REGION Network 64: Step[1390] : Job[13] Step End
   RUNG wire#powerrail
      { S7_Templates := "SrcType := DInt" } EQ_Contact(in1 := "Unit1.Em5.ControlNodes".gaugeRnR.sequence.status.currentStep, in2 := #JOB_13_STEP_90)
      Contact( "Unit1.Em5.ControlNodes".gaugeRnR.sequence.status.seqActive )
      wire#w1
      Coil( "Unit1.Em5.ControlNodes".gaugeRnR."step".action1[1390] )
   END_RUNG
   RUNG wire#w1
      Coil( "Unit1.Em5.ControlNodes".gaugeRnR."step".transition1[1390] )
   END_RUNG
   RUNG wire#w1
      Contact( "Unit1.Em5.ControlNodes".gaugeRnR."step".transition1[1390] )
      Move(in := #STEP_IDLE, out1 => "Unit1.Em5.ControlNodes".gaugeRnR.sequence.status.nextStep)
   END_RUNG
   // the same network as SCL:
   "Unit1.Em5.ControlNodes".gaugeRnR."step".action1[1390] := ("Unit1.Em5.ControlNodes".gaugeRnR.sequence.status.currentStep = #JOB_13_STEP_90) AND "Unit1.Em5.ControlNodes".gaugeRnR.sequence.status.seqActive;
   "Unit1.Em5.ControlNodes".gaugeRnR."step".transition1[1390] := ("Unit1.Em5.ControlNodes".gaugeRnR.sequence.status.currentStep = #JOB_13_STEP_90) AND "Unit1.Em5.ControlNodes".gaugeRnR.sequence.status.seqActive;
   IF ("Unit1.Em5.ControlNodes".gaugeRnR.sequence.status.currentStep = #JOB_13_STEP_90) AND "Unit1.Em5.ControlNodes".gaugeRnR.sequence.status.seqActive AND "Unit1.Em5.ControlNodes".gaugeRnR."step".transition1[1390] THEN
       "Unit1.Em5.ControlNodes".gaugeRnR.sequence.status.nextStep := #STEP_IDLE;
   END_IF;
END_REGION

REGION Network 65: *************** JOB[15] MainPnP Move ReelCut Convyeor / AlignTable************************
END_REGION

REGION Network 66: Step[1501] : Job[15] Condtion
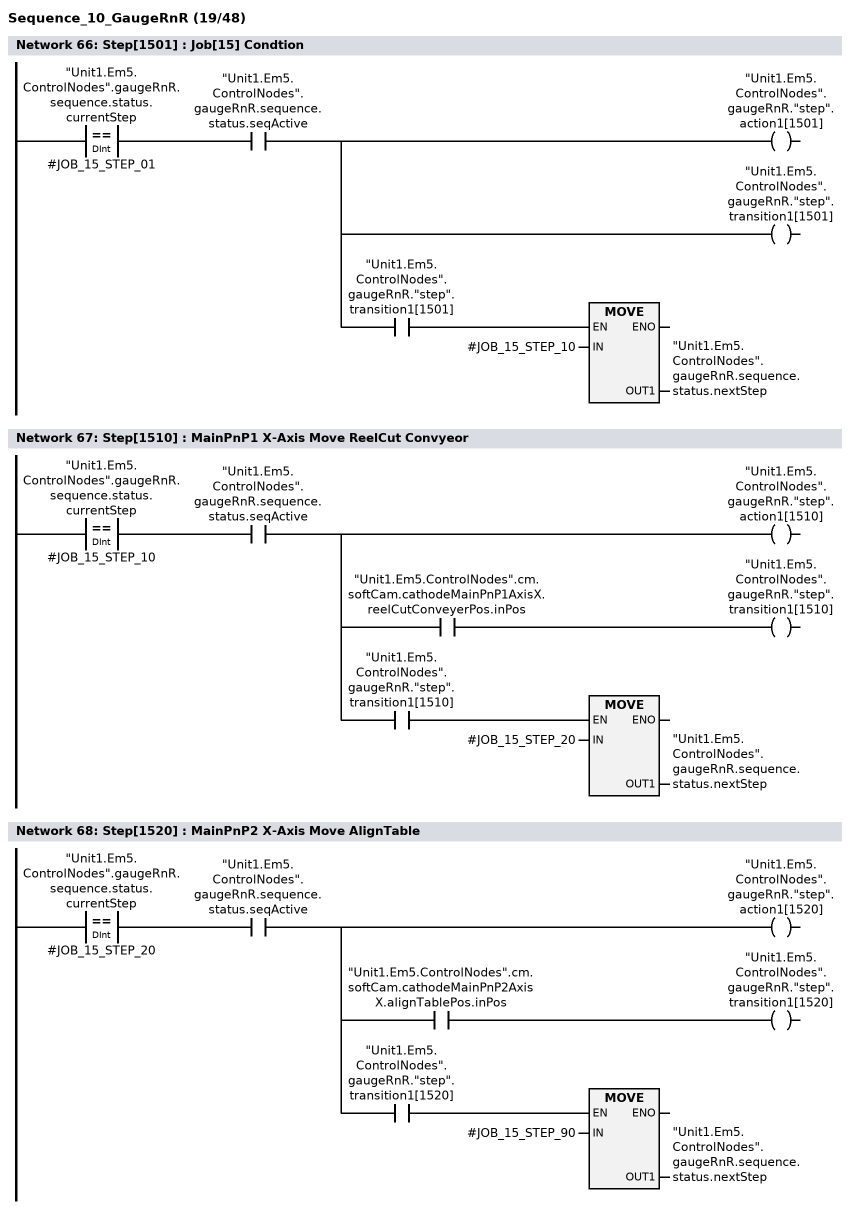
   RUNG wire#powerrail
      { S7_Templates := "SrcType := DInt" } EQ_Contact(in1 := "Unit1.Em5.ControlNodes".gaugeRnR.sequence.status.currentStep, in2 := #JOB_15_STEP_01)
      Contact( "Unit1.Em5.ControlNodes".gaugeRnR.sequence.status.seqActive )
      wire#w1
      Coil( "Unit1.Em5.ControlNodes".gaugeRnR."step".action1[1501] )
   END_RUNG
   RUNG wire#w1
      Coil( "Unit1.Em5.ControlNodes".gaugeRnR."step".transition1[1501] )
   END_RUNG
   RUNG wire#w1
      Contact( "Unit1.Em5.ControlNodes".gaugeRnR."step".transition1[1501] )
      Move(in := #JOB_15_STEP_10, out1 => "Unit1.Em5.ControlNodes".gaugeRnR.sequence.status.nextStep)
   END_RUNG
   // the same network as SCL:
   "Unit1.Em5.ControlNodes".gaugeRnR."step".action1[1501] := ("Unit1.Em5.ControlNodes".gaugeRnR.sequence.status.currentStep = #JOB_15_STEP_01) AND "Unit1.Em5.ControlNodes".gaugeRnR.sequence.status.seqActive;
   "Unit1.Em5.ControlNodes".gaugeRnR."step".transition1[1501] := ("Unit1.Em5.ControlNodes".gaugeRnR.sequence.status.currentStep = #JOB_15_STEP_01) AND "Unit1.Em5.ControlNodes".gaugeRnR.sequence.status.seqActive;
   IF ("Unit1.Em5.ControlNodes".gaugeRnR.sequence.status.currentStep = #JOB_15_STEP_01) AND "Unit1.Em5.ControlNodes".gaugeRnR.sequence.status.seqActive AND "Unit1.Em5.ControlNodes".gaugeRnR."step".transition1[1501] THEN
       "Unit1.Em5.ControlNodes".gaugeRnR.sequence.status.nextStep := #JOB_15_STEP_10;
   END_IF;
END_REGION

REGION Network 67: Step[1510] : MainPnP1 X-Axis Move ReelCut Convyeor
   RUNG wire#powerrail
      { S7_Templates := "SrcType := DInt" } EQ_Contact(in1 := "Unit1.Em5.ControlNodes".gaugeRnR.sequence.status.currentStep, in2 := #JOB_15_STEP_10)
      Contact( "Unit1.Em5.ControlNodes".gaugeRnR.sequence.status.seqActive )
      wire#w1
      Coil( "Unit1.Em5.ControlNodes".gaugeRnR."step".action1[1510] )
   END_RUNG
   RUNG wire#w1
      Contact( "Unit1.Em5.ControlNodes".cm.softCam.cathodeMainPnP1AxisX.reelCutConveyerPos.inPos )
      Coil( "Unit1.Em5.ControlNodes".gaugeRnR."step".transition1[1510] )
   END_RUNG
   RUNG wire#w1
      Contact( "Unit1.Em5.ControlNodes".gaugeRnR."step".transition1[1510] )
      Move(in := #JOB_15_STEP_20, out1 => "Unit1.Em5.ControlNodes".gaugeRnR.sequence.status.nextStep)
   END_RUNG
   // the same network as SCL:
   "Unit1.Em5.ControlNodes".gaugeRnR."step".action1[1510] := ("Unit1.Em5.ControlNodes".gaugeRnR.sequence.status.currentStep = #JOB_15_STEP_10) AND "Unit1.Em5.ControlNodes".gaugeRnR.sequence.status.seqActive;
   "Unit1.Em5.ControlNodes".gaugeRnR."step".transition1[1510] := ("Unit1.Em5.ControlNodes".gaugeRnR.sequence.status.currentStep = #JOB_15_STEP_10) AND "Unit1.Em5.ControlNodes".gaugeRnR.sequence.status.seqActive AND "Unit1.Em5.ControlNodes".cm.softCam.cathodeMainPnP1AxisX.reelCutConveyerPos.inPos;
   IF ("Unit1.Em5.ControlNodes".gaugeRnR.sequence.status.currentStep = #JOB_15_STEP_10) AND "Unit1.Em5.ControlNodes".gaugeRnR.sequence.status.seqActive AND "Unit1.Em5.ControlNodes".gaugeRnR."step".transition1[1510] THEN
       "Unit1.Em5.ControlNodes".gaugeRnR.sequence.status.nextStep := #JOB_15_STEP_20;
   END_IF;
END_REGION

REGION Network 68: Step[1520] : MainPnP2 X-Axis Move AlignTable
   RUNG wire#powerrail
      { S7_Templates := "SrcType := DInt" } EQ_Contact(in1 := "Unit1.Em5.ControlNodes".gaugeRnR.sequence.status.currentStep, in2 := #JOB_15_STEP_20)
      Contact( "Unit1.Em5.ControlNodes".gaugeRnR.sequence.status.seqActive )
      wire#w1
      Coil( "Unit1.Em5.ControlNodes".gaugeRnR."step".action1[1520] )
   END_RUNG
   RUNG wire#w1
      Contact( "Unit1.Em5.ControlNodes".cm.softCam.cathodeMainPnP2AxisX.alignTablePos.inPos )
      Coil( "Unit1.Em5.ControlNodes".gaugeRnR."step".transition1[1520] )
   END_RUNG
   RUNG wire#w1
      Contact( "Unit1.Em5.ControlNodes".gaugeRnR."step".transition1[1520] )
      Move(in := #JOB_15_STEP_90, out1 => "Unit1.Em5.ControlNodes".gaugeRnR.sequence.status.nextStep)
   END_RUNG
   // the same network as SCL:
   "Unit1.Em5.ControlNodes".gaugeRnR."step".action1[1520] := ("Unit1.Em5.ControlNodes".gaugeRnR.sequence.status.currentStep = #JOB_15_STEP_20) AND "Unit1.Em5.ControlNodes".gaugeRnR.sequence.status.seqActive;
   "Unit1.Em5.ControlNodes".gaugeRnR."step".transition1[1520] := ("Unit1.Em5.ControlNodes".gaugeRnR.sequence.status.currentStep = #JOB_15_STEP_20) AND "Unit1.Em5.ControlNodes".gaugeRnR.sequence.status.seqActive AND "Unit1.Em5.ControlNodes".cm.softCam.cathodeMainPnP2AxisX.alignTablePos.inPos;
   IF ("Unit1.Em5.ControlNodes".gaugeRnR.sequence.status.currentStep = #JOB_15_STEP_20) AND "Unit1.Em5.ControlNodes".gaugeRnR.sequence.status.seqActive AND "Unit1.Em5.ControlNodes".gaugeRnR."step".transition1[1520] THEN
       "Unit1.Em5.ControlNodes".gaugeRnR.sequence.status.nextStep := #JOB_15_STEP_90;
   END_IF;
END_REGION

REGION Network 69: Step[1590] : Job[15] Step End
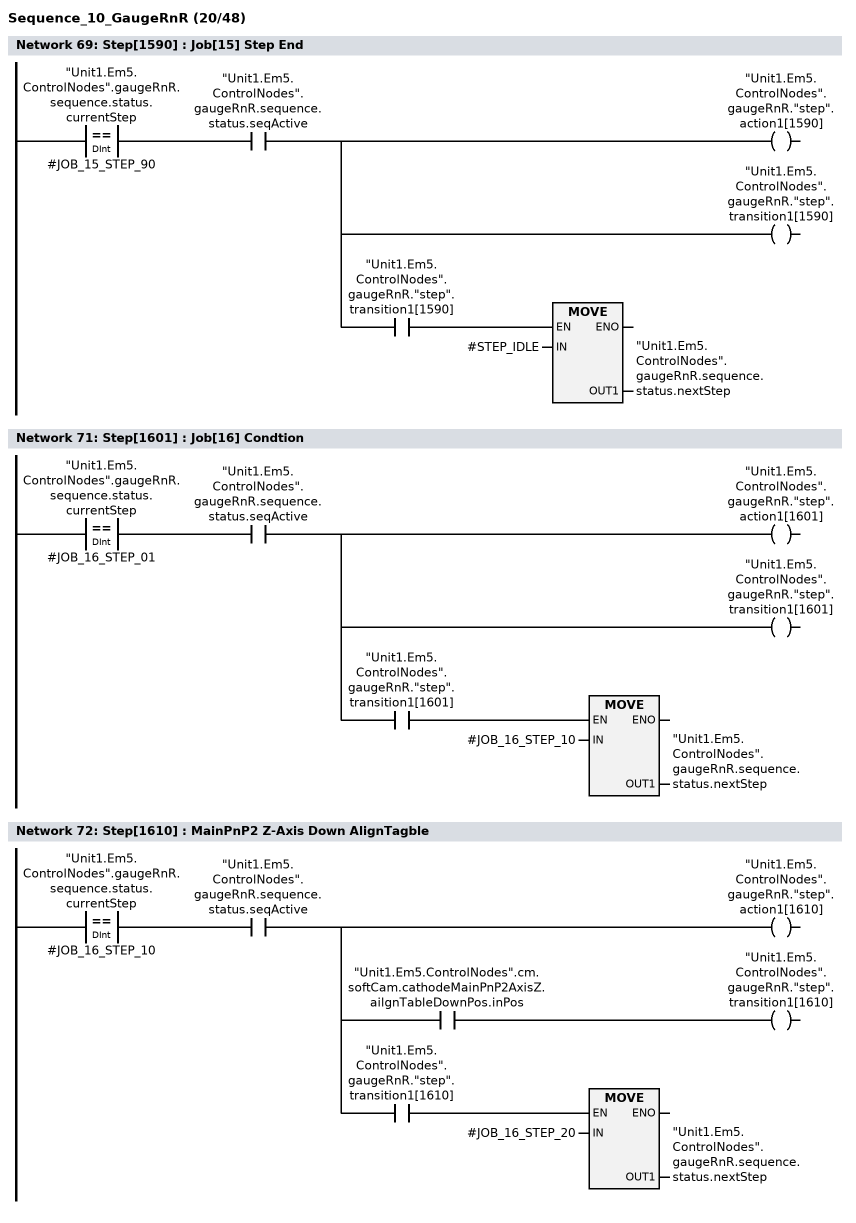
   RUNG wire#powerrail
      { S7_Templates := "SrcType := DInt" } EQ_Contact(in1 := "Unit1.Em5.ControlNodes".gaugeRnR.sequence.status.currentStep, in2 := #JOB_15_STEP_90)
      Contact( "Unit1.Em5.ControlNodes".gaugeRnR.sequence.status.seqActive )
      wire#w1
      Coil( "Unit1.Em5.ControlNodes".gaugeRnR."step".action1[1590] )
   END_RUNG
   RUNG wire#w1
      Coil( "Unit1.Em5.ControlNodes".gaugeRnR."step".transition1[1590] )
   END_RUNG
   RUNG wire#w1
      Contact( "Unit1.Em5.ControlNodes".gaugeRnR."step".transition1[1590] )
      Move(in := #STEP_IDLE, out1 => "Unit1.Em5.ControlNodes".gaugeRnR.sequence.status.nextStep)
   END_RUNG
   // the same network as SCL:
   "Unit1.Em5.ControlNodes".gaugeRnR."step".action1[1590] := ("Unit1.Em5.ControlNodes".gaugeRnR.sequence.status.currentStep = #JOB_15_STEP_90) AND "Unit1.Em5.ControlNodes".gaugeRnR.sequence.status.seqActive;
   "Unit1.Em5.ControlNodes".gaugeRnR."step".transition1[1590] := ("Unit1.Em5.ControlNodes".gaugeRnR.sequence.status.currentStep = #JOB_15_STEP_90) AND "Unit1.Em5.ControlNodes".gaugeRnR.sequence.status.seqActive;
   IF ("Unit1.Em5.ControlNodes".gaugeRnR.sequence.status.currentStep = #JOB_15_STEP_90) AND "Unit1.Em5.ControlNodes".gaugeRnR.sequence.status.seqActive AND "Unit1.Em5.ControlNodes".gaugeRnR."step".transition1[1590] THEN
       "Unit1.Em5.ControlNodes".gaugeRnR.sequence.status.nextStep := #STEP_IDLE;
   END_IF;
END_REGION

REGION Network 70: *************** JOB[16] AlignTable To MainPnP2 ************************
END_REGION

REGION Network 71: Step[1601] : Job[16] Condtion
   RUNG wire#powerrail
      { S7_Templates := "SrcType := DInt" } EQ_Contact(in1 := "Unit1.Em5.ControlNodes".gaugeRnR.sequence.status.currentStep, in2 := #JOB_16_STEP_01)
      Contact( "Unit1.Em5.ControlNodes".gaugeRnR.sequence.status.seqActive )
      wire#w1
      Coil( "Unit1.Em5.ControlNodes".gaugeRnR."step".action1[1601] )
   END_RUNG
   RUNG wire#w1
      Coil( "Unit1.Em5.ControlNodes".gaugeRnR."step".transition1[1601] )
   END_RUNG
   RUNG wire#w1
      Contact( "Unit1.Em5.ControlNodes".gaugeRnR."step".transition1[1601] )
      Move(in := #JOB_16_STEP_10, out1 => "Unit1.Em5.ControlNodes".gaugeRnR.sequence.status.nextStep)
   END_RUNG
   // the same network as SCL:
   "Unit1.Em5.ControlNodes".gaugeRnR."step".action1[1601] := ("Unit1.Em5.ControlNodes".gaugeRnR.sequence.status.currentStep = #JOB_16_STEP_01) AND "Unit1.Em5.ControlNodes".gaugeRnR.sequence.status.seqActive;
   "Unit1.Em5.ControlNodes".gaugeRnR."step".transition1[1601] := ("Unit1.Em5.ControlNodes".gaugeRnR.sequence.status.currentStep = #JOB_16_STEP_01) AND "Unit1.Em5.ControlNodes".gaugeRnR.sequence.status.seqActive;
   IF ("Unit1.Em5.ControlNodes".gaugeRnR.sequence.status.currentStep = #JOB_16_STEP_01) AND "Unit1.Em5.ControlNodes".gaugeRnR.sequence.status.seqActive AND "Unit1.Em5.ControlNodes".gaugeRnR."step".transition1[1601] THEN
       "Unit1.Em5.ControlNodes".gaugeRnR.sequence.status.nextStep := #JOB_16_STEP_10;
   END_IF;
END_REGION

REGION Network 72: Step[1610] : MainPnP2 Z-Axis Down AlignTagble
   RUNG wire#powerrail
      { S7_Templates := "SrcType := DInt" } EQ_Contact(in1 := "Unit1.Em5.ControlNodes".gaugeRnR.sequence.status.currentStep, in2 := #JOB_16_STEP_10)
      Contact( "Unit1.Em5.ControlNodes".gaugeRnR.sequence.status.seqActive )
      wire#w1
      Coil( "Unit1.Em5.ControlNodes".gaugeRnR."step".action1[1610] )
   END_RUNG
   RUNG wire#w1
      Contact( "Unit1.Em5.ControlNodes".cm.softCam.cathodeMainPnP2AxisZ.ailgnTableDownPos.inPos )
      Coil( "Unit1.Em5.ControlNodes".gaugeRnR."step".transition1[1610] )
   END_RUNG
   RUNG wire#w1
      Contact( "Unit1.Em5.ControlNodes".gaugeRnR."step".transition1[1610] )
      Move(in := #JOB_16_STEP_20, out1 => "Unit1.Em5.ControlNodes".gaugeRnR.sequence.status.nextStep)
   END_RUNG
   // the same network as SCL:
   "Unit1.Em5.ControlNodes".gaugeRnR."step".action1[1610] := ("Unit1.Em5.ControlNodes".gaugeRnR.sequence.status.currentStep = #JOB_16_STEP_10) AND "Unit1.Em5.ControlNodes".gaugeRnR.sequence.status.seqActive;
   "Unit1.Em5.ControlNodes".gaugeRnR."step".transition1[1610] := ("Unit1.Em5.ControlNodes".gaugeRnR.sequence.status.currentStep = #JOB_16_STEP_10) AND "Unit1.Em5.ControlNodes".gaugeRnR.sequence.status.seqActive AND "Unit1.Em5.ControlNodes".cm.softCam.cathodeMainPnP2AxisZ.ailgnTableDownPos.inPos;
   IF ("Unit1.Em5.ControlNodes".gaugeRnR.sequence.status.currentStep = #JOB_16_STEP_10) AND "Unit1.Em5.ControlNodes".gaugeRnR.sequence.status.seqActive AND "Unit1.Em5.ControlNodes".gaugeRnR."step".transition1[1610] THEN
       "Unit1.Em5.ControlNodes".gaugeRnR.sequence.status.nextStep := #JOB_16_STEP_20;
   END_IF;
END_REGION

REGION Network 73: Step[1620] : AlignTable Vaccum Off
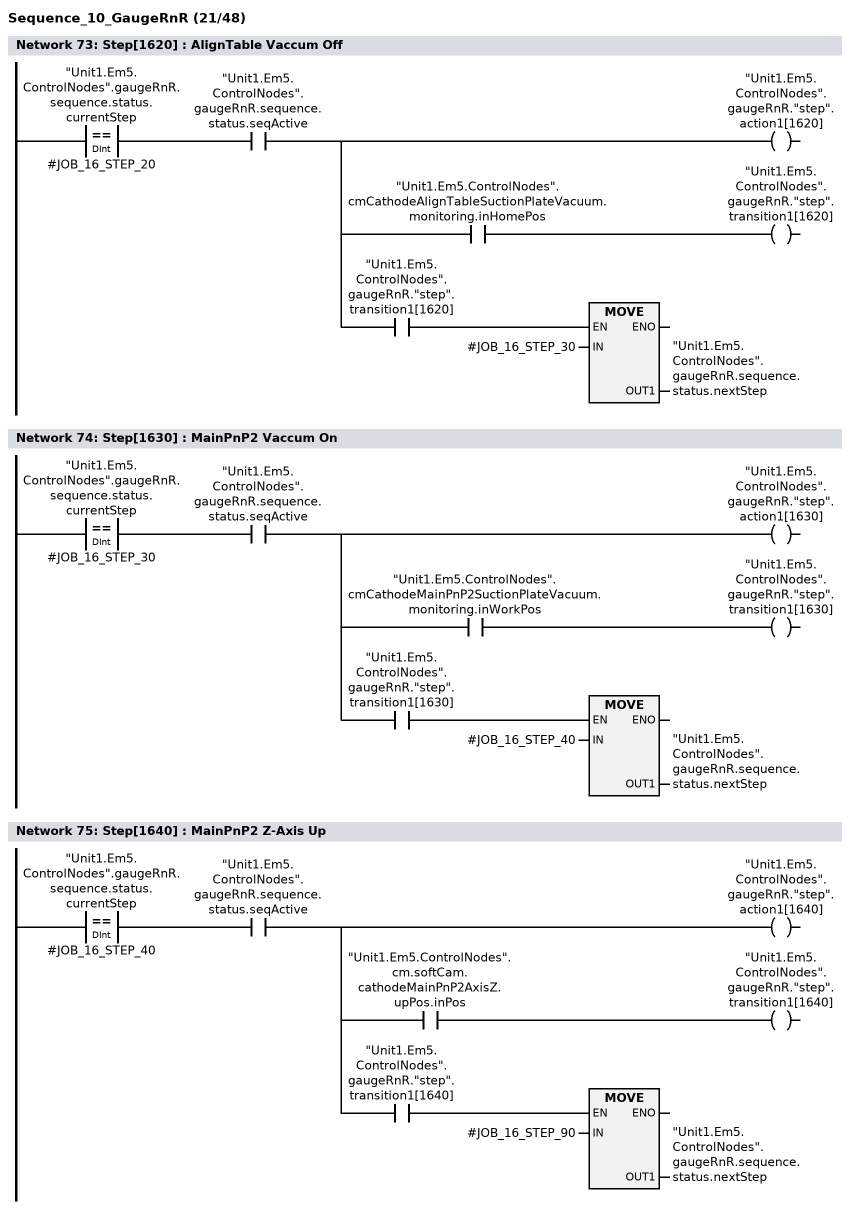
   RUNG wire#powerrail
      { S7_Templates := "SrcType := DInt" } EQ_Contact(in1 := "Unit1.Em5.ControlNodes".gaugeRnR.sequence.status.currentStep, in2 := #JOB_16_STEP_20)
      Contact( "Unit1.Em5.ControlNodes".gaugeRnR.sequence.status.seqActive )
      wire#w1
      Coil( "Unit1.Em5.ControlNodes".gaugeRnR."step".action1[1620] )
   END_RUNG
   RUNG wire#w1
      Contact( "Unit1.Em5.ControlNodes".cmCathodeAlignTableSuctionPlateVacuum.monitoring.inHomePos )
      Coil( "Unit1.Em5.ControlNodes".gaugeRnR."step".transition1[1620] )
   END_RUNG
   RUNG wire#w1
      Contact( "Unit1.Em5.ControlNodes".gaugeRnR."step".transition1[1620] )
      Move(in := #JOB_16_STEP_30, out1 => "Unit1.Em5.ControlNodes".gaugeRnR.sequence.status.nextStep)
   END_RUNG
   // the same network as SCL:
   "Unit1.Em5.ControlNodes".gaugeRnR."step".action1[1620] := ("Unit1.Em5.ControlNodes".gaugeRnR.sequence.status.currentStep = #JOB_16_STEP_20) AND "Unit1.Em5.ControlNodes".gaugeRnR.sequence.status.seqActive;
   "Unit1.Em5.ControlNodes".gaugeRnR."step".transition1[1620] := ("Unit1.Em5.ControlNodes".gaugeRnR.sequence.status.currentStep = #JOB_16_STEP_20) AND "Unit1.Em5.ControlNodes".gaugeRnR.sequence.status.seqActive AND "Unit1.Em5.ControlNodes".cmCathodeAlignTableSuctionPlateVacuum.monitoring.inHomePos;
   IF ("Unit1.Em5.ControlNodes".gaugeRnR.sequence.status.currentStep = #JOB_16_STEP_20) AND "Unit1.Em5.ControlNodes".gaugeRnR.sequence.status.seqActive AND "Unit1.Em5.ControlNodes".gaugeRnR."step".transition1[1620] THEN
       "Unit1.Em5.ControlNodes".gaugeRnR.sequence.status.nextStep := #JOB_16_STEP_30;
   END_IF;
END_REGION

REGION Network 74: Step[1630] : MainPnP2 Vaccum On
   RUNG wire#powerrail
      { S7_Templates := "SrcType := DInt" } EQ_Contact(in1 := "Unit1.Em5.ControlNodes".gaugeRnR.sequence.status.currentStep, in2 := #JOB_16_STEP_30)
      Contact( "Unit1.Em5.ControlNodes".gaugeRnR.sequence.status.seqActive )
      wire#w1
      Coil( "Unit1.Em5.ControlNodes".gaugeRnR."step".action1[1630] )
   END_RUNG
   RUNG wire#w1
      Contact( "Unit1.Em5.ControlNodes".cmCathodeMainPnP2SuctionPlateVacuum.monitoring.inWorkPos )
      Coil( "Unit1.Em5.ControlNodes".gaugeRnR."step".transition1[1630] )
   END_RUNG
   RUNG wire#w1
      Contact( "Unit1.Em5.ControlNodes".gaugeRnR."step".transition1[1630] )
      Move(in := #JOB_16_STEP_40, out1 => "Unit1.Em5.ControlNodes".gaugeRnR.sequence.status.nextStep)
   END_RUNG
   // the same network as SCL:
   "Unit1.Em5.ControlNodes".gaugeRnR."step".action1[1630] := ("Unit1.Em5.ControlNodes".gaugeRnR.sequence.status.currentStep = #JOB_16_STEP_30) AND "Unit1.Em5.ControlNodes".gaugeRnR.sequence.status.seqActive;
   "Unit1.Em5.ControlNodes".gaugeRnR."step".transition1[1630] := ("Unit1.Em5.ControlNodes".gaugeRnR.sequence.status.currentStep = #JOB_16_STEP_30) AND "Unit1.Em5.ControlNodes".gaugeRnR.sequence.status.seqActive AND "Unit1.Em5.ControlNodes".cmCathodeMainPnP2SuctionPlateVacuum.monitoring.inWorkPos;
   IF ("Unit1.Em5.ControlNodes".gaugeRnR.sequence.status.currentStep = #JOB_16_STEP_30) AND "Unit1.Em5.ControlNodes".gaugeRnR.sequence.status.seqActive AND "Unit1.Em5.ControlNodes".gaugeRnR."step".transition1[1630] THEN
       "Unit1.Em5.ControlNodes".gaugeRnR.sequence.status.nextStep := #JOB_16_STEP_40;
   END_IF;
END_REGION

REGION Network 75: Step[1640] : MainPnP2 Z-Axis Up
   RUNG wire#powerrail
      { S7_Templates := "SrcType := DInt" } EQ_Contact(in1 := "Unit1.Em5.ControlNodes".gaugeRnR.sequence.status.currentStep, in2 := #JOB_16_STEP_40)
      Contact( "Unit1.Em5.ControlNodes".gaugeRnR.sequence.status.seqActive )
      wire#w1
      Coil( "Unit1.Em5.ControlNodes".gaugeRnR."step".action1[1640] )
   END_RUNG
   RUNG wire#w1
      Contact( "Unit1.Em5.ControlNodes".cm.softCam.cathodeMainPnP2AxisZ.upPos.inPos )
      Coil( "Unit1.Em5.ControlNodes".gaugeRnR."step".transition1[1640] )
   END_RUNG
   RUNG wire#w1
      Contact( "Unit1.Em5.ControlNodes".gaugeRnR."step".transition1[1640] )
      Move(in := #JOB_16_STEP_90, out1 => "Unit1.Em5.ControlNodes".gaugeRnR.sequence.status.nextStep)
   END_RUNG
   // the same network as SCL:
   "Unit1.Em5.ControlNodes".gaugeRnR."step".action1[1640] := ("Unit1.Em5.ControlNodes".gaugeRnR.sequence.status.currentStep = #JOB_16_STEP_40) AND "Unit1.Em5.ControlNodes".gaugeRnR.sequence.status.seqActive;
   "Unit1.Em5.ControlNodes".gaugeRnR."step".transition1[1640] := ("Unit1.Em5.ControlNodes".gaugeRnR.sequence.status.currentStep = #JOB_16_STEP_40) AND "Unit1.Em5.ControlNodes".gaugeRnR.sequence.status.seqActive AND "Unit1.Em5.ControlNodes".cm.softCam.cathodeMainPnP2AxisZ.upPos.inPos;
   IF ("Unit1.Em5.ControlNodes".gaugeRnR.sequence.status.currentStep = #JOB_16_STEP_40) AND "Unit1.Em5.ControlNodes".gaugeRnR.sequence.status.seqActive AND "Unit1.Em5.ControlNodes".gaugeRnR."step".transition1[1640] THEN
       "Unit1.Em5.ControlNodes".gaugeRnR.sequence.status.nextStep := #JOB_16_STEP_90;
   END_IF;
END_REGION

REGION Network 76: Step[1690] : Job[16] Step End
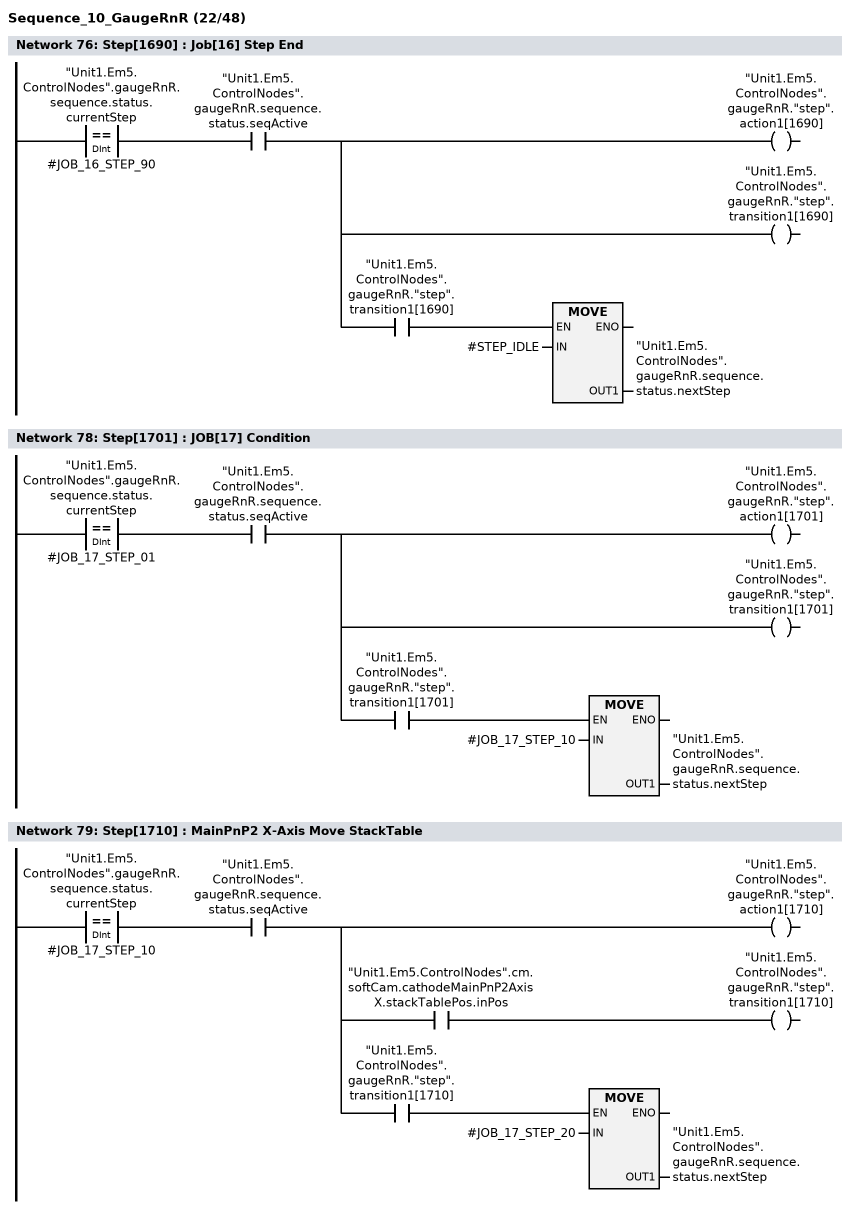
   RUNG wire#powerrail
      { S7_Templates := "SrcType := DInt" } EQ_Contact(in1 := "Unit1.Em5.ControlNodes".gaugeRnR.sequence.status.currentStep, in2 := #JOB_16_STEP_90)
      Contact( "Unit1.Em5.ControlNodes".gaugeRnR.sequence.status.seqActive )
      wire#w1
      Coil( "Unit1.Em5.ControlNodes".gaugeRnR."step".action1[1690] )
   END_RUNG
   RUNG wire#w1
      Coil( "Unit1.Em5.ControlNodes".gaugeRnR."step".transition1[1690] )
   END_RUNG
   RUNG wire#w1
      Contact( "Unit1.Em5.ControlNodes".gaugeRnR."step".transition1[1690] )
      Move(in := #STEP_IDLE, out1 => "Unit1.Em5.ControlNodes".gaugeRnR.sequence.status.nextStep)
   END_RUNG
   // the same network as SCL:
   "Unit1.Em5.ControlNodes".gaugeRnR."step".action1[1690] := ("Unit1.Em5.ControlNodes".gaugeRnR.sequence.status.currentStep = #JOB_16_STEP_90) AND "Unit1.Em5.ControlNodes".gaugeRnR.sequence.status.seqActive;
   "Unit1.Em5.ControlNodes".gaugeRnR."step".transition1[1690] := ("Unit1.Em5.ControlNodes".gaugeRnR.sequence.status.currentStep = #JOB_16_STEP_90) AND "Unit1.Em5.ControlNodes".gaugeRnR.sequence.status.seqActive;
   IF ("Unit1.Em5.ControlNodes".gaugeRnR.sequence.status.currentStep = #JOB_16_STEP_90) AND "Unit1.Em5.ControlNodes".gaugeRnR.sequence.status.seqActive AND "Unit1.Em5.ControlNodes".gaugeRnR."step".transition1[1690] THEN
       "Unit1.Em5.ControlNodes".gaugeRnR.sequence.status.nextStep := #STEP_IDLE;
   END_IF;
END_REGION

REGION Network 77: *************** JOB[17] MainPnP Move AlignTable / StackTable ************************
END_REGION

REGION Network 78: Step[1701] : JOB[17] Condition
   RUNG wire#powerrail
      { S7_Templates := "SrcType := DInt" } EQ_Contact(in1 := "Unit1.Em5.ControlNodes".gaugeRnR.sequence.status.currentStep, in2 := #JOB_17_STEP_01)
      Contact( "Unit1.Em5.ControlNodes".gaugeRnR.sequence.status.seqActive )
      wire#w1
      Coil( "Unit1.Em5.ControlNodes".gaugeRnR."step".action1[1701] )
   END_RUNG
   RUNG wire#w1
      Coil( "Unit1.Em5.ControlNodes".gaugeRnR."step".transition1[1701] )
   END_RUNG
   RUNG wire#w1
      Contact( "Unit1.Em5.ControlNodes".gaugeRnR."step".transition1[1701] )
      Move(in := #JOB_17_STEP_10, out1 => "Unit1.Em5.ControlNodes".gaugeRnR.sequence.status.nextStep)
   END_RUNG
   // the same network as SCL:
   "Unit1.Em5.ControlNodes".gaugeRnR."step".action1[1701] := ("Unit1.Em5.ControlNodes".gaugeRnR.sequence.status.currentStep = #JOB_17_STEP_01) AND "Unit1.Em5.ControlNodes".gaugeRnR.sequence.status.seqActive;
   "Unit1.Em5.ControlNodes".gaugeRnR."step".transition1[1701] := ("Unit1.Em5.ControlNodes".gaugeRnR.sequence.status.currentStep = #JOB_17_STEP_01) AND "Unit1.Em5.ControlNodes".gaugeRnR.sequence.status.seqActive;
   IF ("Unit1.Em5.ControlNodes".gaugeRnR.sequence.status.currentStep = #JOB_17_STEP_01) AND "Unit1.Em5.ControlNodes".gaugeRnR.sequence.status.seqActive AND "Unit1.Em5.ControlNodes".gaugeRnR."step".transition1[1701] THEN
       "Unit1.Em5.ControlNodes".gaugeRnR.sequence.status.nextStep := #JOB_17_STEP_10;
   END_IF;
END_REGION

REGION Network 79: Step[1710] : MainPnP2 X-Axis Move StackTable
   RUNG wire#powerrail
      { S7_Templates := "SrcType := DInt" } EQ_Contact(in1 := "Unit1.Em5.ControlNodes".gaugeRnR.sequence.status.currentStep, in2 := #JOB_17_STEP_10)
      Contact( "Unit1.Em5.ControlNodes".gaugeRnR.sequence.status.seqActive )
      wire#w1
      Coil( "Unit1.Em5.ControlNodes".gaugeRnR."step".action1[1710] )
   END_RUNG
   RUNG wire#w1
      Contact( "Unit1.Em5.ControlNodes".cm.softCam.cathodeMainPnP2AxisX.stackTablePos.inPos )
      Coil( "Unit1.Em5.ControlNodes".gaugeRnR."step".transition1[1710] )
   END_RUNG
   RUNG wire#w1
      Contact( "Unit1.Em5.ControlNodes".gaugeRnR."step".transition1[1710] )
      Move(in := #JOB_17_STEP_20, out1 => "Unit1.Em5.ControlNodes".gaugeRnR.sequence.status.nextStep)
   END_RUNG
   // the same network as SCL:
   "Unit1.Em5.ControlNodes".gaugeRnR."step".action1[1710] := ("Unit1.Em5.ControlNodes".gaugeRnR.sequence.status.currentStep = #JOB_17_STEP_10) AND "Unit1.Em5.ControlNodes".gaugeRnR.sequence.status.seqActive;
   "Unit1.Em5.ControlNodes".gaugeRnR."step".transition1[1710] := ("Unit1.Em5.ControlNodes".gaugeRnR.sequence.status.currentStep = #JOB_17_STEP_10) AND "Unit1.Em5.ControlNodes".gaugeRnR.sequence.status.seqActive AND "Unit1.Em5.ControlNodes".cm.softCam.cathodeMainPnP2AxisX.stackTablePos.inPos;
   IF ("Unit1.Em5.ControlNodes".gaugeRnR.sequence.status.currentStep = #JOB_17_STEP_10) AND "Unit1.Em5.ControlNodes".gaugeRnR.sequence.status.seqActive AND "Unit1.Em5.ControlNodes".gaugeRnR."step".transition1[1710] THEN
       "Unit1.Em5.ControlNodes".gaugeRnR.sequence.status.nextStep := #JOB_17_STEP_20;
   END_IF;
END_REGION

REGION Network 80: Step[1720] : MainPnP1 X-Axis Move AlignTable
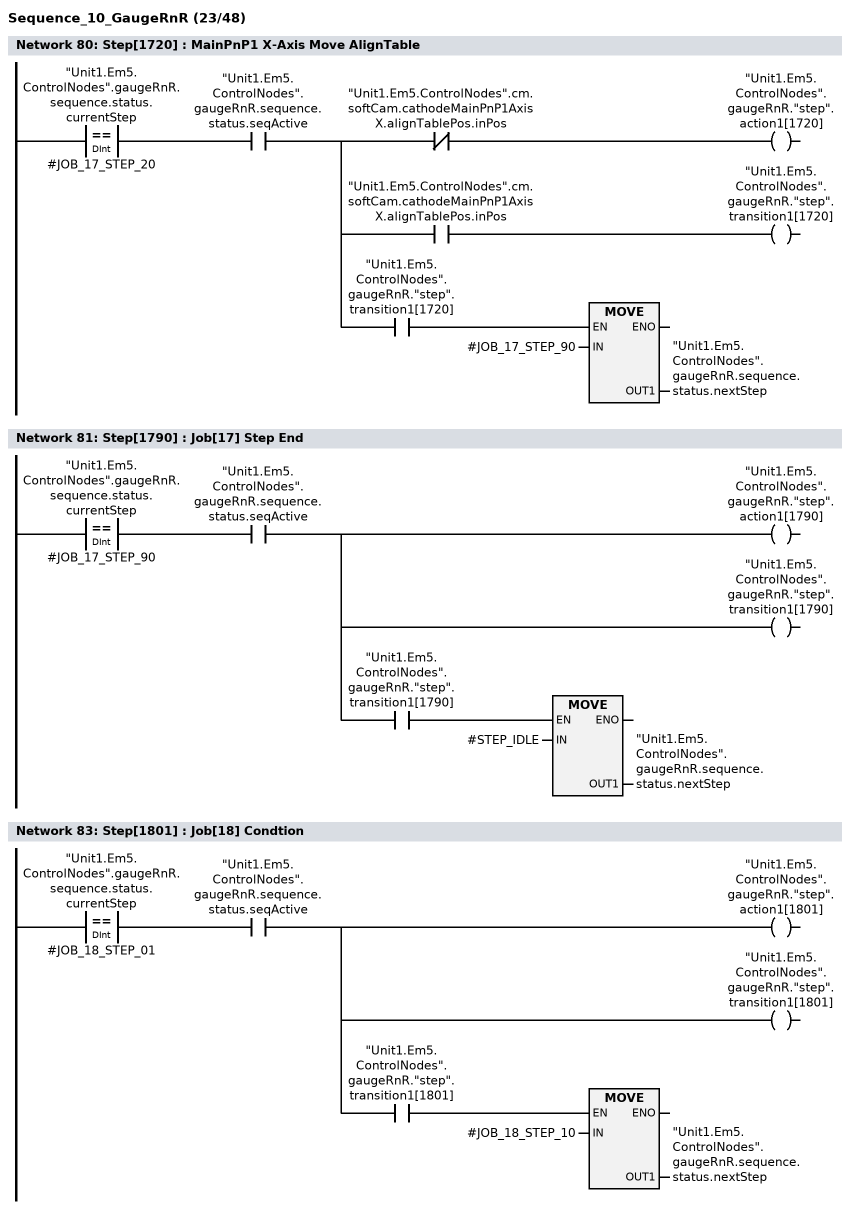
   RUNG wire#powerrail
      { S7_Templates := "SrcType := DInt" } EQ_Contact(in1 := "Unit1.Em5.ControlNodes".gaugeRnR.sequence.status.currentStep, in2 := #JOB_17_STEP_20)
      Contact( "Unit1.Em5.ControlNodes".gaugeRnR.sequence.status.seqActive )
      wire#w1
      I_Contact( "Unit1.Em5.ControlNodes".cm.softCam.cathodeMainPnP1AxisX.alignTablePos.inPos )
      Coil( "Unit1.Em5.ControlNodes".gaugeRnR."step".action1[1720] )
   END_RUNG
   RUNG wire#w1
      Contact( "Unit1.Em5.ControlNodes".cm.softCam.cathodeMainPnP1AxisX.alignTablePos.inPos )
      Coil( "Unit1.Em5.ControlNodes".gaugeRnR."step".transition1[1720] )
   END_RUNG
   RUNG wire#w1
      Contact( "Unit1.Em5.ControlNodes".gaugeRnR."step".transition1[1720] )
      Move(in := #JOB_17_STEP_90, out1 => "Unit1.Em5.ControlNodes".gaugeRnR.sequence.status.nextStep)
   END_RUNG
   // the same network as SCL:
   #_w1 := ("Unit1.Em5.ControlNodes".gaugeRnR.sequence.status.currentStep = #JOB_17_STEP_20) AND "Unit1.Em5.ControlNodes".gaugeRnR.sequence.status.seqActive;
   "Unit1.Em5.ControlNodes".gaugeRnR."step".action1[1720] := #_w1 AND NOT "Unit1.Em5.ControlNodes".cm.softCam.cathodeMainPnP1AxisX.alignTablePos.inPos;
   "Unit1.Em5.ControlNodes".gaugeRnR."step".transition1[1720] := #_w1 AND "Unit1.Em5.ControlNodes".cm.softCam.cathodeMainPnP1AxisX.alignTablePos.inPos;
   IF #_w1 AND "Unit1.Em5.ControlNodes".gaugeRnR."step".transition1[1720] THEN
       "Unit1.Em5.ControlNodes".gaugeRnR.sequence.status.nextStep := #JOB_17_STEP_90;
   END_IF;
END_REGION

REGION Network 81: Step[1790] : Job[17] Step End
   RUNG wire#powerrail
      { S7_Templates := "SrcType := DInt" } EQ_Contact(in1 := "Unit1.Em5.ControlNodes".gaugeRnR.sequence.status.currentStep, in2 := #JOB_17_STEP_90)
      Contact( "Unit1.Em5.ControlNodes".gaugeRnR.sequence.status.seqActive )
      wire#w1
      Coil( "Unit1.Em5.ControlNodes".gaugeRnR."step".action1[1790] )
   END_RUNG
   RUNG wire#w1
      Coil( "Unit1.Em5.ControlNodes".gaugeRnR."step".transition1[1790] )
   END_RUNG
   RUNG wire#w1
      Contact( "Unit1.Em5.ControlNodes".gaugeRnR."step".transition1[1790] )
      Move(in := #STEP_IDLE, out1 => "Unit1.Em5.ControlNodes".gaugeRnR.sequence.status.nextStep)
   END_RUNG
   // the same network as SCL:
   "Unit1.Em5.ControlNodes".gaugeRnR."step".action1[1790] := ("Unit1.Em5.ControlNodes".gaugeRnR.sequence.status.currentStep = #JOB_17_STEP_90) AND "Unit1.Em5.ControlNodes".gaugeRnR.sequence.status.seqActive;
   "Unit1.Em5.ControlNodes".gaugeRnR."step".transition1[1790] := ("Unit1.Em5.ControlNodes".gaugeRnR.sequence.status.currentStep = #JOB_17_STEP_90) AND "Unit1.Em5.ControlNodes".gaugeRnR.sequence.status.seqActive;
   IF ("Unit1.Em5.ControlNodes".gaugeRnR.sequence.status.currentStep = #JOB_17_STEP_90) AND "Unit1.Em5.ControlNodes".gaugeRnR.sequence.status.seqActive AND "Unit1.Em5.ControlNodes".gaugeRnR."step".transition1[1790] THEN
       "Unit1.Em5.ControlNodes".gaugeRnR.sequence.status.nextStep := #STEP_IDLE;
   END_IF;
END_REGION

REGION Network 82: *************** JOB[18] AlignTable Move Wait ************************
END_REGION

REGION Network 83: Step[1801] : Job[18] Condtion
   RUNG wire#powerrail
      { S7_Templates := "SrcType := DInt" } EQ_Contact(in1 := "Unit1.Em5.ControlNodes".gaugeRnR.sequence.status.currentStep, in2 := #JOB_18_STEP_01)
      Contact( "Unit1.Em5.ControlNodes".gaugeRnR.sequence.status.seqActive )
      wire#w1
      Coil( "Unit1.Em5.ControlNodes".gaugeRnR."step".action1[1801] )
   END_RUNG
   RUNG wire#w1
      Coil( "Unit1.Em5.ControlNodes".gaugeRnR."step".transition1[1801] )
   END_RUNG
   RUNG wire#w1
      Contact( "Unit1.Em5.ControlNodes".gaugeRnR."step".transition1[1801] )
      Move(in := #JOB_18_STEP_10, out1 => "Unit1.Em5.ControlNodes".gaugeRnR.sequence.status.nextStep)
   END_RUNG
   // the same network as SCL:
   "Unit1.Em5.ControlNodes".gaugeRnR."step".action1[1801] := ("Unit1.Em5.ControlNodes".gaugeRnR.sequence.status.currentStep = #JOB_18_STEP_01) AND "Unit1.Em5.ControlNodes".gaugeRnR.sequence.status.seqActive;
   "Unit1.Em5.ControlNodes".gaugeRnR."step".transition1[1801] := ("Unit1.Em5.ControlNodes".gaugeRnR.sequence.status.currentStep = #JOB_18_STEP_01) AND "Unit1.Em5.ControlNodes".gaugeRnR.sequence.status.seqActive;
   IF ("Unit1.Em5.ControlNodes".gaugeRnR.sequence.status.currentStep = #JOB_18_STEP_01) AND "Unit1.Em5.ControlNodes".gaugeRnR.sequence.status.seqActive AND "Unit1.Em5.ControlNodes".gaugeRnR."step".transition1[1801] THEN
       "Unit1.Em5.ControlNodes".gaugeRnR.sequence.status.nextStep := #JOB_18_STEP_10;
   END_IF;
END_REGION

REGION Network 84: Step[1810] : AlignTable Move Wait
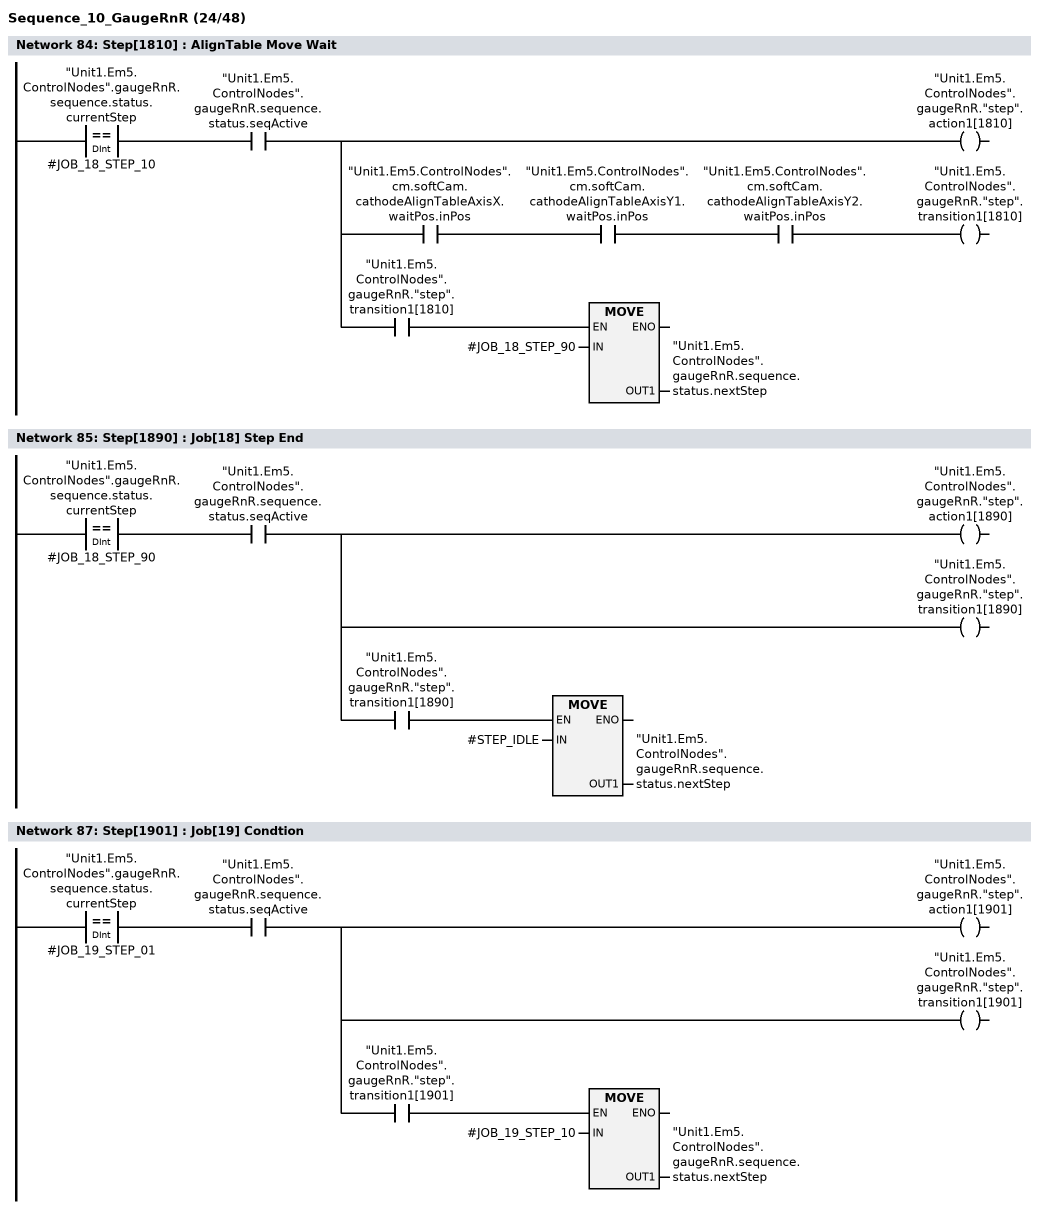
   RUNG wire#powerrail
      { S7_Templates := "SrcType := DInt" } EQ_Contact(in1 := "Unit1.Em5.ControlNodes".gaugeRnR.sequence.status.currentStep, in2 := #JOB_18_STEP_10)
      Contact( "Unit1.Em5.ControlNodes".gaugeRnR.sequence.status.seqActive )
      wire#w1
      Coil( "Unit1.Em5.ControlNodes".gaugeRnR."step".action1[1810] )
   END_RUNG
   RUNG wire#w1
      Contact( "Unit1.Em5.ControlNodes".cm.softCam.cathodeAlignTableAxisX.waitPos.inPos )
      Contact( "Unit1.Em5.ControlNodes".cm.softCam.cathodeAlignTableAxisY1.waitPos.inPos )
      Contact( "Unit1.Em5.ControlNodes".cm.softCam.cathodeAlignTableAxisY2.waitPos.inPos )
      Coil( "Unit1.Em5.ControlNodes".gaugeRnR."step".transition1[1810] )
   END_RUNG
   RUNG wire#w1
      Contact( "Unit1.Em5.ControlNodes".gaugeRnR."step".transition1[1810] )
      Move(in := #JOB_18_STEP_90, out1 => "Unit1.Em5.ControlNodes".gaugeRnR.sequence.status.nextStep)
   END_RUNG
   // the same network as SCL:
   "Unit1.Em5.ControlNodes".gaugeRnR."step".action1[1810] := ("Unit1.Em5.ControlNodes".gaugeRnR.sequence.status.currentStep = #JOB_18_STEP_10) AND "Unit1.Em5.ControlNodes".gaugeRnR.sequence.status.seqActive;
   "Unit1.Em5.ControlNodes".gaugeRnR."step".transition1[1810] := ("Unit1.Em5.ControlNodes".gaugeRnR.sequence.status.currentStep = #JOB_18_STEP_10) AND "Unit1.Em5.ControlNodes".gaugeRnR.sequence.status.seqActive AND "Unit1.Em5.ControlNodes".cm.softCam.cathodeAlignTableAxisX.waitPos.inPos AND "Unit1.Em5.ControlNodes".cm.softCam.cathodeAlignTableAxisY1.waitPos.inPos AND "Unit1.Em5.ControlNodes".cm.softCam.cathodeAlignTableAxisY2.waitPos.inPos;
   IF ("Unit1.Em5.ControlNodes".gaugeRnR.sequence.status.currentStep = #JOB_18_STEP_10) AND "Unit1.Em5.ControlNodes".gaugeRnR.sequence.status.seqActive AND "Unit1.Em5.ControlNodes".gaugeRnR."step".transition1[1810] THEN
       "Unit1.Em5.ControlNodes".gaugeRnR.sequence.status.nextStep := #JOB_18_STEP_90;
   END_IF;
END_REGION

REGION Network 85: Step[1890] : Job[18] Step End
   RUNG wire#powerrail
      { S7_Templates := "SrcType := DInt" } EQ_Contact(in1 := "Unit1.Em5.ControlNodes".gaugeRnR.sequence.status.currentStep, in2 := #JOB_18_STEP_90)
      Contact( "Unit1.Em5.ControlNodes".gaugeRnR.sequence.status.seqActive )
      wire#w1
      Coil( "Unit1.Em5.ControlNodes".gaugeRnR."step".action1[1890] )
   END_RUNG
   RUNG wire#w1
      Coil( "Unit1.Em5.ControlNodes".gaugeRnR."step".transition1[1890] )
   END_RUNG
   RUNG wire#w1
      Contact( "Unit1.Em5.ControlNodes".gaugeRnR."step".transition1[1890] )
      Move(in := #STEP_IDLE, out1 => "Unit1.Em5.ControlNodes".gaugeRnR.sequence.status.nextStep)
   END_RUNG
   // the same network as SCL:
   "Unit1.Em5.ControlNodes".gaugeRnR."step".action1[1890] := ("Unit1.Em5.ControlNodes".gaugeRnR.sequence.status.currentStep = #JOB_18_STEP_90) AND "Unit1.Em5.ControlNodes".gaugeRnR.sequence.status.seqActive;
   "Unit1.Em5.ControlNodes".gaugeRnR."step".transition1[1890] := ("Unit1.Em5.ControlNodes".gaugeRnR.sequence.status.currentStep = #JOB_18_STEP_90) AND "Unit1.Em5.ControlNodes".gaugeRnR.sequence.status.seqActive;
   IF ("Unit1.Em5.ControlNodes".gaugeRnR.sequence.status.currentStep = #JOB_18_STEP_90) AND "Unit1.Em5.ControlNodes".gaugeRnR.sequence.status.seqActive AND "Unit1.Em5.ControlNodes".gaugeRnR."step".transition1[1890] THEN
       "Unit1.Em5.ControlNodes".gaugeRnR.sequence.status.nextStep := #STEP_IDLE;
   END_IF;
END_REGION

REGION Network 86: *************** JOB[19] MainPnP2 To StackTable ************************
END_REGION

REGION Network 87: Step[1901] : Job[19] Condtion
   RUNG wire#powerrail
      { S7_Templates := "SrcType := DInt" } EQ_Contact(in1 := "Unit1.Em5.ControlNodes".gaugeRnR.sequence.status.currentStep, in2 := #JOB_19_STEP_01)
      Contact( "Unit1.Em5.ControlNodes".gaugeRnR.sequence.status.seqActive )
      wire#w1
      Coil( "Unit1.Em5.ControlNodes".gaugeRnR."step".action1[1901] )
   END_RUNG
   RUNG wire#w1
      Coil( "Unit1.Em5.ControlNodes".gaugeRnR."step".transition1[1901] )
   END_RUNG
   RUNG wire#w1
      Contact( "Unit1.Em5.ControlNodes".gaugeRnR."step".transition1[1901] )
      Move(in := #JOB_19_STEP_10, out1 => "Unit1.Em5.ControlNodes".gaugeRnR.sequence.status.nextStep)
   END_RUNG
   // the same network as SCL:
   "Unit1.Em5.ControlNodes".gaugeRnR."step".action1[1901] := ("Unit1.Em5.ControlNodes".gaugeRnR.sequence.status.currentStep = #JOB_19_STEP_01) AND "Unit1.Em5.ControlNodes".gaugeRnR.sequence.status.seqActive;
   "Unit1.Em5.ControlNodes".gaugeRnR."step".transition1[1901] := ("Unit1.Em5.ControlNodes".gaugeRnR.sequence.status.currentStep = #JOB_19_STEP_01) AND "Unit1.Em5.ControlNodes".gaugeRnR.sequence.status.seqActive;
   IF ("Unit1.Em5.ControlNodes".gaugeRnR.sequence.status.currentStep = #JOB_19_STEP_01) AND "Unit1.Em5.ControlNodes".gaugeRnR.sequence.status.seqActive AND "Unit1.Em5.ControlNodes".gaugeRnR."step".transition1[1901] THEN
       "Unit1.Em5.ControlNodes".gaugeRnR.sequence.status.nextStep := #JOB_19_STEP_10;
   END_IF;
END_REGION

REGION Network 88: Step[1910] : MainPnP2 Z-Axis Move StackTable Down
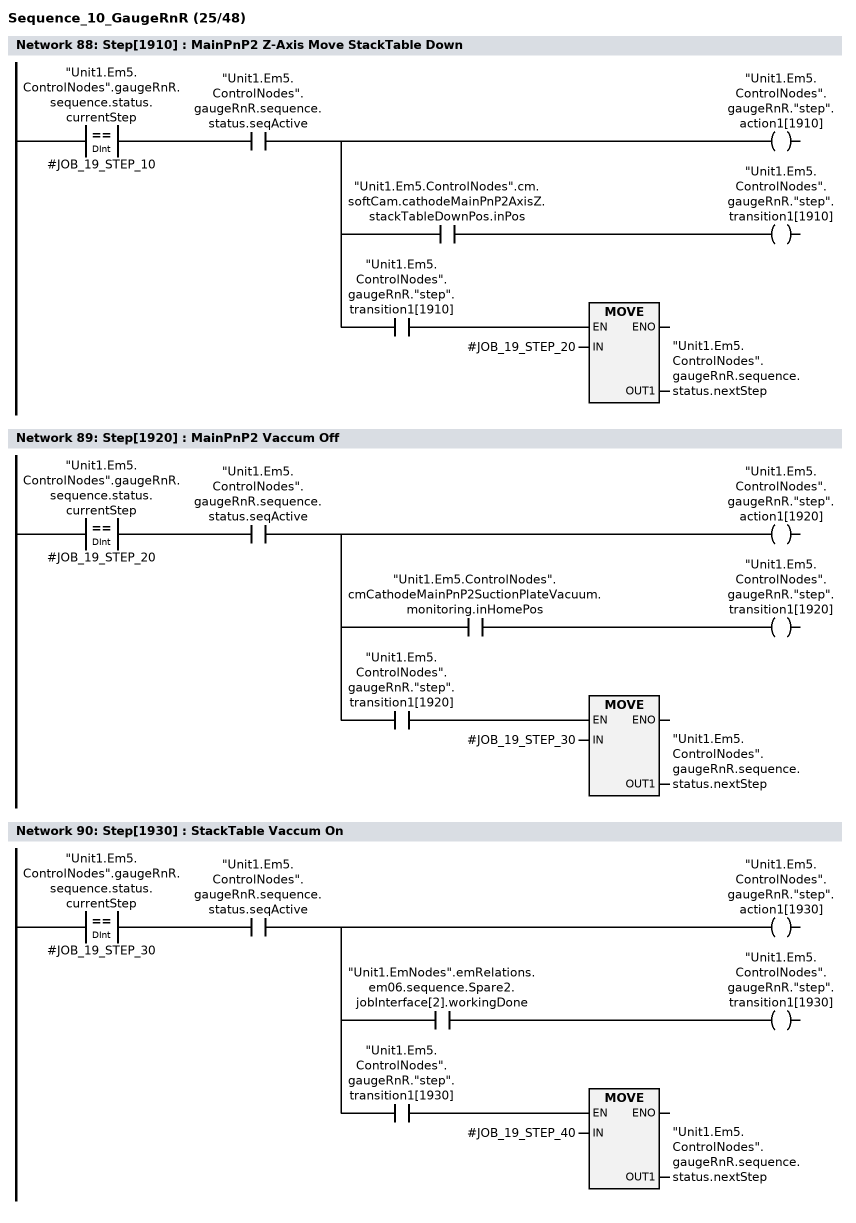
   RUNG wire#powerrail
      { S7_Templates := "SrcType := DInt" } EQ_Contact(in1 := "Unit1.Em5.ControlNodes".gaugeRnR.sequence.status.currentStep, in2 := #JOB_19_STEP_10)
      Contact( "Unit1.Em5.ControlNodes".gaugeRnR.sequence.status.seqActive )
      wire#w1
      Coil( "Unit1.Em5.ControlNodes".gaugeRnR."step".action1[1910] )
   END_RUNG
   RUNG wire#w1
      Contact( "Unit1.Em5.ControlNodes".cm.softCam.cathodeMainPnP2AxisZ.stackTableDownPos.inPos )
      Coil( "Unit1.Em5.ControlNodes".gaugeRnR."step".transition1[1910] )
   END_RUNG
   RUNG wire#w1
      Contact( "Unit1.Em5.ControlNodes".gaugeRnR."step".transition1[1910] )
      Move(in := #JOB_19_STEP_20, out1 => "Unit1.Em5.ControlNodes".gaugeRnR.sequence.status.nextStep)
   END_RUNG
   // the same network as SCL:
   "Unit1.Em5.ControlNodes".gaugeRnR."step".action1[1910] := ("Unit1.Em5.ControlNodes".gaugeRnR.sequence.status.currentStep = #JOB_19_STEP_10) AND "Unit1.Em5.ControlNodes".gaugeRnR.sequence.status.seqActive;
   "Unit1.Em5.ControlNodes".gaugeRnR."step".transition1[1910] := ("Unit1.Em5.ControlNodes".gaugeRnR.sequence.status.currentStep = #JOB_19_STEP_10) AND "Unit1.Em5.ControlNodes".gaugeRnR.sequence.status.seqActive AND "Unit1.Em5.ControlNodes".cm.softCam.cathodeMainPnP2AxisZ.stackTableDownPos.inPos;
   IF ("Unit1.Em5.ControlNodes".gaugeRnR.sequence.status.currentStep = #JOB_19_STEP_10) AND "Unit1.Em5.ControlNodes".gaugeRnR.sequence.status.seqActive AND "Unit1.Em5.ControlNodes".gaugeRnR."step".transition1[1910] THEN
       "Unit1.Em5.ControlNodes".gaugeRnR.sequence.status.nextStep := #JOB_19_STEP_20;
   END_IF;
END_REGION

REGION Network 89: Step[1920] : MainPnP2 Vaccum Off
   RUNG wire#powerrail
      { S7_Templates := "SrcType := DInt" } EQ_Contact(in1 := "Unit1.Em5.ControlNodes".gaugeRnR.sequence.status.currentStep, in2 := #JOB_19_STEP_20)
      Contact( "Unit1.Em5.ControlNodes".gaugeRnR.sequence.status.seqActive )
      wire#w1
      Coil( "Unit1.Em5.ControlNodes".gaugeRnR."step".action1[1920] )
   END_RUNG
   RUNG wire#w1
      Contact( "Unit1.Em5.ControlNodes".cmCathodeMainPnP2SuctionPlateVacuum.monitoring.inHomePos )
      Coil( "Unit1.Em5.ControlNodes".gaugeRnR."step".transition1[1920] )
   END_RUNG
   RUNG wire#w1
      Contact( "Unit1.Em5.ControlNodes".gaugeRnR."step".transition1[1920] )
      Move(in := #JOB_19_STEP_30, out1 => "Unit1.Em5.ControlNodes".gaugeRnR.sequence.status.nextStep)
   END_RUNG
   // the same network as SCL:
   "Unit1.Em5.ControlNodes".gaugeRnR."step".action1[1920] := ("Unit1.Em5.ControlNodes".gaugeRnR.sequence.status.currentStep = #JOB_19_STEP_20) AND "Unit1.Em5.ControlNodes".gaugeRnR.sequence.status.seqActive;
   "Unit1.Em5.ControlNodes".gaugeRnR."step".transition1[1920] := ("Unit1.Em5.ControlNodes".gaugeRnR.sequence.status.currentStep = #JOB_19_STEP_20) AND "Unit1.Em5.ControlNodes".gaugeRnR.sequence.status.seqActive AND "Unit1.Em5.ControlNodes".cmCathodeMainPnP2SuctionPlateVacuum.monitoring.inHomePos;
   IF ("Unit1.Em5.ControlNodes".gaugeRnR.sequence.status.currentStep = #JOB_19_STEP_20) AND "Unit1.Em5.ControlNodes".gaugeRnR.sequence.status.seqActive AND "Unit1.Em5.ControlNodes".gaugeRnR."step".transition1[1920] THEN
       "Unit1.Em5.ControlNodes".gaugeRnR.sequence.status.nextStep := #JOB_19_STEP_30;
   END_IF;
END_REGION

REGION Network 90: Step[1930] : StackTable Vaccum On
   RUNG wire#powerrail
      { S7_Templates := "SrcType := DInt" } EQ_Contact(in1 := "Unit1.Em5.ControlNodes".gaugeRnR.sequence.status.currentStep, in2 := #JOB_19_STEP_30)
      Contact( "Unit1.Em5.ControlNodes".gaugeRnR.sequence.status.seqActive )
      wire#w1
      Coil( "Unit1.Em5.ControlNodes".gaugeRnR."step".action1[1930] )
   END_RUNG
   RUNG wire#w1
      Contact( "Unit1.EmNodes".emRelations.em06.sequence.Spare2.jobInterface[2].workingDone )
      Coil( "Unit1.Em5.ControlNodes".gaugeRnR."step".transition1[1930] )
   END_RUNG
   RUNG wire#w1
      Contact( "Unit1.Em5.ControlNodes".gaugeRnR."step".transition1[1930] )
      Move(in := #JOB_19_STEP_40, out1 => "Unit1.Em5.ControlNodes".gaugeRnR.sequence.status.nextStep)
   END_RUNG
   // the same network as SCL:
   "Unit1.Em5.ControlNodes".gaugeRnR."step".action1[1930] := ("Unit1.Em5.ControlNodes".gaugeRnR.sequence.status.currentStep = #JOB_19_STEP_30) AND "Unit1.Em5.ControlNodes".gaugeRnR.sequence.status.seqActive;
   "Unit1.Em5.ControlNodes".gaugeRnR."step".transition1[1930] := ("Unit1.Em5.ControlNodes".gaugeRnR.sequence.status.currentStep = #JOB_19_STEP_30) AND "Unit1.Em5.ControlNodes".gaugeRnR.sequence.status.seqActive AND "Unit1.EmNodes".emRelations.em06.sequence.Spare2.jobInterface[2].workingDone;
   IF ("Unit1.Em5.ControlNodes".gaugeRnR.sequence.status.currentStep = #JOB_19_STEP_30) AND "Unit1.Em5.ControlNodes".gaugeRnR.sequence.status.seqActive AND "Unit1.Em5.ControlNodes".gaugeRnR."step".transition1[1930] THEN
       "Unit1.Em5.ControlNodes".gaugeRnR.sequence.status.nextStep := #JOB_19_STEP_40;
   END_IF;
END_REGION

REGION Network 91: Step[1940] : MainPnP2 Z-Axis Up
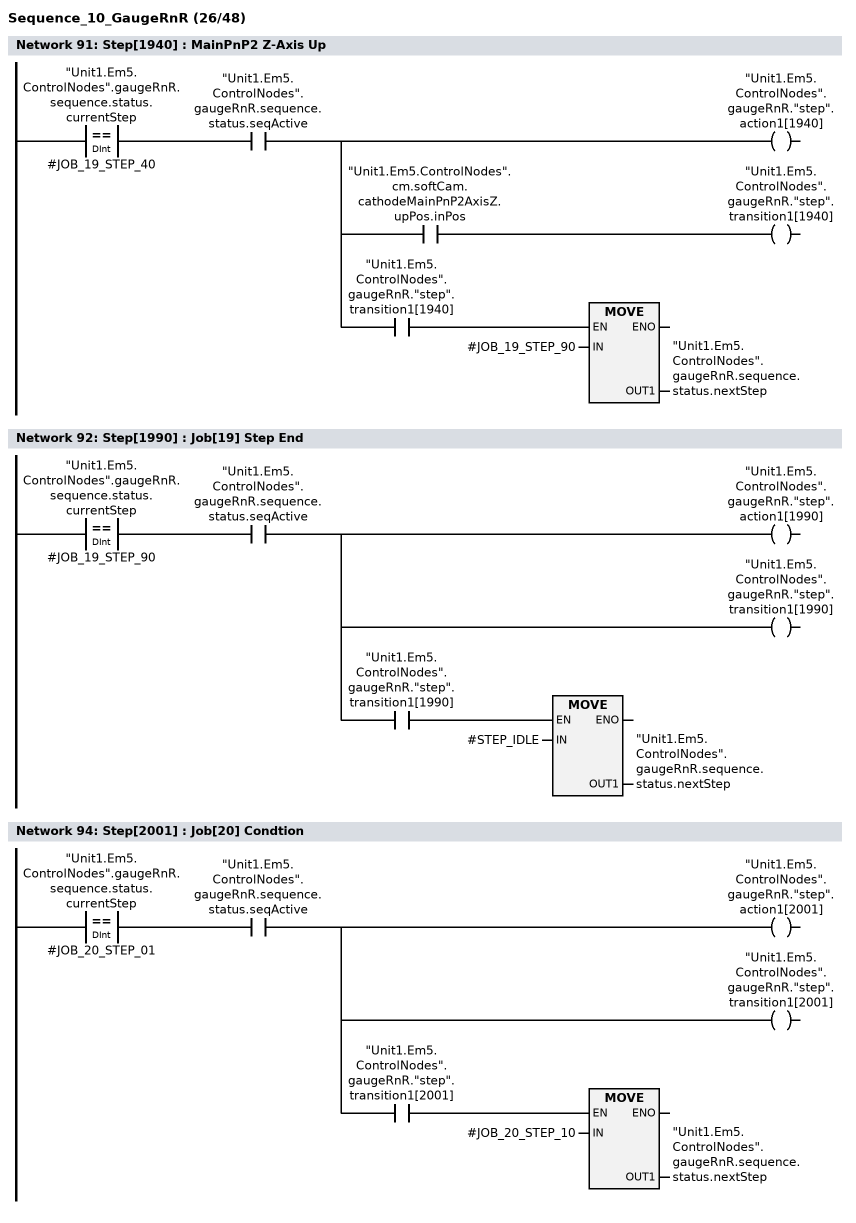
   RUNG wire#powerrail
      { S7_Templates := "SrcType := DInt" } EQ_Contact(in1 := "Unit1.Em5.ControlNodes".gaugeRnR.sequence.status.currentStep, in2 := #JOB_19_STEP_40)
      Contact( "Unit1.Em5.ControlNodes".gaugeRnR.sequence.status.seqActive )
      wire#w1
      Coil( "Unit1.Em5.ControlNodes".gaugeRnR."step".action1[1940] )
   END_RUNG
   RUNG wire#w1
      Contact( "Unit1.Em5.ControlNodes".cm.softCam.cathodeMainPnP2AxisZ.upPos.inPos )
      Coil( "Unit1.Em5.ControlNodes".gaugeRnR."step".transition1[1940] )
   END_RUNG
   RUNG wire#w1
      Contact( "Unit1.Em5.ControlNodes".gaugeRnR."step".transition1[1940] )
      Move(in := #JOB_19_STEP_90, out1 => "Unit1.Em5.ControlNodes".gaugeRnR.sequence.status.nextStep)
   END_RUNG
   // the same network as SCL:
   "Unit1.Em5.ControlNodes".gaugeRnR."step".action1[1940] := ("Unit1.Em5.ControlNodes".gaugeRnR.sequence.status.currentStep = #JOB_19_STEP_40) AND "Unit1.Em5.ControlNodes".gaugeRnR.sequence.status.seqActive;
   "Unit1.Em5.ControlNodes".gaugeRnR."step".transition1[1940] := ("Unit1.Em5.ControlNodes".gaugeRnR.sequence.status.currentStep = #JOB_19_STEP_40) AND "Unit1.Em5.ControlNodes".gaugeRnR.sequence.status.seqActive AND "Unit1.Em5.ControlNodes".cm.softCam.cathodeMainPnP2AxisZ.upPos.inPos;
   IF ("Unit1.Em5.ControlNodes".gaugeRnR.sequence.status.currentStep = #JOB_19_STEP_40) AND "Unit1.Em5.ControlNodes".gaugeRnR.sequence.status.seqActive AND "Unit1.Em5.ControlNodes".gaugeRnR."step".transition1[1940] THEN
       "Unit1.Em5.ControlNodes".gaugeRnR.sequence.status.nextStep := #JOB_19_STEP_90;
   END_IF;
END_REGION

REGION Network 92: Step[1990] : Job[19] Step End
   RUNG wire#powerrail
      { S7_Templates := "SrcType := DInt" } EQ_Contact(in1 := "Unit1.Em5.ControlNodes".gaugeRnR.sequence.status.currentStep, in2 := #JOB_19_STEP_90)
      Contact( "Unit1.Em5.ControlNodes".gaugeRnR.sequence.status.seqActive )
      wire#w1
      Coil( "Unit1.Em5.ControlNodes".gaugeRnR."step".action1[1990] )
   END_RUNG
   RUNG wire#w1
      Coil( "Unit1.Em5.ControlNodes".gaugeRnR."step".transition1[1990] )
   END_RUNG
   RUNG wire#w1
      Contact( "Unit1.Em5.ControlNodes".gaugeRnR."step".transition1[1990] )
      Move(in := #STEP_IDLE, out1 => "Unit1.Em5.ControlNodes".gaugeRnR.sequence.status.nextStep)
   END_RUNG
   // the same network as SCL:
   "Unit1.Em5.ControlNodes".gaugeRnR."step".action1[1990] := ("Unit1.Em5.ControlNodes".gaugeRnR.sequence.status.currentStep = #JOB_19_STEP_90) AND "Unit1.Em5.ControlNodes".gaugeRnR.sequence.status.seqActive;
   "Unit1.Em5.ControlNodes".gaugeRnR."step".transition1[1990] := ("Unit1.Em5.ControlNodes".gaugeRnR.sequence.status.currentStep = #JOB_19_STEP_90) AND "Unit1.Em5.ControlNodes".gaugeRnR.sequence.status.seqActive;
   IF ("Unit1.Em5.ControlNodes".gaugeRnR.sequence.status.currentStep = #JOB_19_STEP_90) AND "Unit1.Em5.ControlNodes".gaugeRnR.sequence.status.seqActive AND "Unit1.Em5.ControlNodes".gaugeRnR."step".transition1[1990] THEN
       "Unit1.Em5.ControlNodes".gaugeRnR.sequence.status.nextStep := #STEP_IDLE;
   END_IF;
END_REGION

REGION Network 93: *************** JOB[20] StackTable To MainPnP2 ************************
END_REGION

REGION Network 94: Step[2001] : Job[20] Condtion
   RUNG wire#powerrail
      { S7_Templates := "SrcType := DInt" } EQ_Contact(in1 := "Unit1.Em5.ControlNodes".gaugeRnR.sequence.status.currentStep, in2 := #JOB_20_STEP_01)
      Contact( "Unit1.Em5.ControlNodes".gaugeRnR.sequence.status.seqActive )
      wire#w1
      Coil( "Unit1.Em5.ControlNodes".gaugeRnR."step".action1[2001] )
   END_RUNG
   RUNG wire#w1
      Coil( "Unit1.Em5.ControlNodes".gaugeRnR."step".transition1[2001] )
   END_RUNG
   RUNG wire#w1
      Contact( "Unit1.Em5.ControlNodes".gaugeRnR."step".transition1[2001] )
      Move(in := #JOB_20_STEP_10, out1 => "Unit1.Em5.ControlNodes".gaugeRnR.sequence.status.nextStep)
   END_RUNG
   // the same network as SCL:
   "Unit1.Em5.ControlNodes".gaugeRnR."step".action1[2001] := ("Unit1.Em5.ControlNodes".gaugeRnR.sequence.status.currentStep = #JOB_20_STEP_01) AND "Unit1.Em5.ControlNodes".gaugeRnR.sequence.status.seqActive;
   "Unit1.Em5.ControlNodes".gaugeRnR."step".transition1[2001] := ("Unit1.Em5.ControlNodes".gaugeRnR.sequence.status.currentStep = #JOB_20_STEP_01) AND "Unit1.Em5.ControlNodes".gaugeRnR.sequence.status.seqActive;
   IF ("Unit1.Em5.ControlNodes".gaugeRnR.sequence.status.currentStep = #JOB_20_STEP_01) AND "Unit1.Em5.ControlNodes".gaugeRnR.sequence.status.seqActive AND "Unit1.Em5.ControlNodes".gaugeRnR."step".transition1[2001] THEN
       "Unit1.Em5.ControlNodes".gaugeRnR.sequence.status.nextStep := #JOB_20_STEP_10;
   END_IF;
END_REGION

REGION Network 95: Step[2010] : MainPnP2 Z-Axis Move StackTable Down
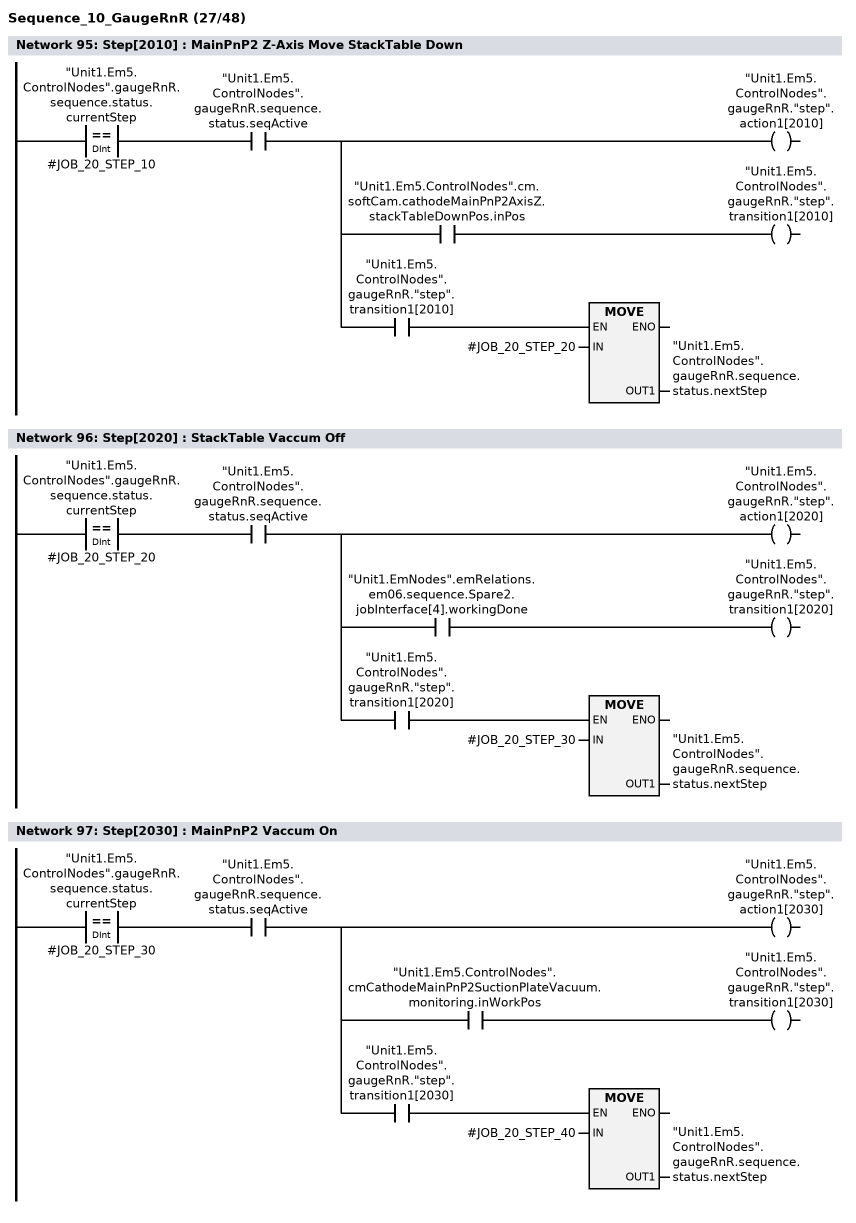
   RUNG wire#powerrail
      { S7_Templates := "SrcType := DInt" } EQ_Contact(in1 := "Unit1.Em5.ControlNodes".gaugeRnR.sequence.status.currentStep, in2 := #JOB_20_STEP_10)
      Contact( "Unit1.Em5.ControlNodes".gaugeRnR.sequence.status.seqActive )
      wire#w1
      Coil( "Unit1.Em5.ControlNodes".gaugeRnR."step".action1[2010] )
   END_RUNG
   RUNG wire#w1
      Contact( "Unit1.Em5.ControlNodes".cm.softCam.cathodeMainPnP2AxisZ.stackTableDownPos.inPos )
      Coil( "Unit1.Em5.ControlNodes".gaugeRnR."step".transition1[2010] )
   END_RUNG
   RUNG wire#w1
      Contact( "Unit1.Em5.ControlNodes".gaugeRnR."step".transition1[2010] )
      Move(in := #JOB_20_STEP_20, out1 => "Unit1.Em5.ControlNodes".gaugeRnR.sequence.status.nextStep)
   END_RUNG
   // the same network as SCL:
   "Unit1.Em5.ControlNodes".gaugeRnR."step".action1[2010] := ("Unit1.Em5.ControlNodes".gaugeRnR.sequence.status.currentStep = #JOB_20_STEP_10) AND "Unit1.Em5.ControlNodes".gaugeRnR.sequence.status.seqActive;
   "Unit1.Em5.ControlNodes".gaugeRnR."step".transition1[2010] := ("Unit1.Em5.ControlNodes".gaugeRnR.sequence.status.currentStep = #JOB_20_STEP_10) AND "Unit1.Em5.ControlNodes".gaugeRnR.sequence.status.seqActive AND "Unit1.Em5.ControlNodes".cm.softCam.cathodeMainPnP2AxisZ.stackTableDownPos.inPos;
   IF ("Unit1.Em5.ControlNodes".gaugeRnR.sequence.status.currentStep = #JOB_20_STEP_10) AND "Unit1.Em5.ControlNodes".gaugeRnR.sequence.status.seqActive AND "Unit1.Em5.ControlNodes".gaugeRnR."step".transition1[2010] THEN
       "Unit1.Em5.ControlNodes".gaugeRnR.sequence.status.nextStep := #JOB_20_STEP_20;
   END_IF;
END_REGION

REGION Network 96: Step[2020] : StackTable Vaccum Off
   RUNG wire#powerrail
      { S7_Templates := "SrcType := DInt" } EQ_Contact(in1 := "Unit1.Em5.ControlNodes".gaugeRnR.sequence.status.currentStep, in2 := #JOB_20_STEP_20)
      Contact( "Unit1.Em5.ControlNodes".gaugeRnR.sequence.status.seqActive )
      wire#w1
      Coil( "Unit1.Em5.ControlNodes".gaugeRnR."step".action1[2020] )
   END_RUNG
   RUNG wire#w1
      Contact( "Unit1.EmNodes".emRelations.em06.sequence.Spare2.jobInterface[4].workingDone )
      Coil( "Unit1.Em5.ControlNodes".gaugeRnR."step".transition1[2020] )
   END_RUNG
   RUNG wire#w1
      Contact( "Unit1.Em5.ControlNodes".gaugeRnR."step".transition1[2020] )
      Move(in := #JOB_20_STEP_30, out1 => "Unit1.Em5.ControlNodes".gaugeRnR.sequence.status.nextStep)
   END_RUNG
   // the same network as SCL:
   "Unit1.Em5.ControlNodes".gaugeRnR."step".action1[2020] := ("Unit1.Em5.ControlNodes".gaugeRnR.sequence.status.currentStep = #JOB_20_STEP_20) AND "Unit1.Em5.ControlNodes".gaugeRnR.sequence.status.seqActive;
   "Unit1.Em5.ControlNodes".gaugeRnR."step".transition1[2020] := ("Unit1.Em5.ControlNodes".gaugeRnR.sequence.status.currentStep = #JOB_20_STEP_20) AND "Unit1.Em5.ControlNodes".gaugeRnR.sequence.status.seqActive AND "Unit1.EmNodes".emRelations.em06.sequence.Spare2.jobInterface[4].workingDone;
   IF ("Unit1.Em5.ControlNodes".gaugeRnR.sequence.status.currentStep = #JOB_20_STEP_20) AND "Unit1.Em5.ControlNodes".gaugeRnR.sequence.status.seqActive AND "Unit1.Em5.ControlNodes".gaugeRnR."step".transition1[2020] THEN
       "Unit1.Em5.ControlNodes".gaugeRnR.sequence.status.nextStep := #JOB_20_STEP_30;
   END_IF;
END_REGION

REGION Network 97: Step[2030] : MainPnP2 Vaccum On
   RUNG wire#powerrail
      { S7_Templates := "SrcType := DInt" } EQ_Contact(in1 := "Unit1.Em5.ControlNodes".gaugeRnR.sequence.status.currentStep, in2 := #JOB_20_STEP_30)
      Contact( "Unit1.Em5.ControlNodes".gaugeRnR.sequence.status.seqActive )
      wire#w1
      Coil( "Unit1.Em5.ControlNodes".gaugeRnR."step".action1[2030] )
   END_RUNG
   RUNG wire#w1
      Contact( "Unit1.Em5.ControlNodes".cmCathodeMainPnP2SuctionPlateVacuum.monitoring.inWorkPos )
      Coil( "Unit1.Em5.ControlNodes".gaugeRnR."step".transition1[2030] )
   END_RUNG
   RUNG wire#w1
      Contact( "Unit1.Em5.ControlNodes".gaugeRnR."step".transition1[2030] )
      Move(in := #JOB_20_STEP_40, out1 => "Unit1.Em5.ControlNodes".gaugeRnR.sequence.status.nextStep)
   END_RUNG
   // the same network as SCL:
   "Unit1.Em5.ControlNodes".gaugeRnR."step".action1[2030] := ("Unit1.Em5.ControlNodes".gaugeRnR.sequence.status.currentStep = #JOB_20_STEP_30) AND "Unit1.Em5.ControlNodes".gaugeRnR.sequence.status.seqActive;
   "Unit1.Em5.ControlNodes".gaugeRnR."step".transition1[2030] := ("Unit1.Em5.ControlNodes".gaugeRnR.sequence.status.currentStep = #JOB_20_STEP_30) AND "Unit1.Em5.ControlNodes".gaugeRnR.sequence.status.seqActive AND "Unit1.Em5.ControlNodes".cmCathodeMainPnP2SuctionPlateVacuum.monitoring.inWorkPos;
   IF ("Unit1.Em5.ControlNodes".gaugeRnR.sequence.status.currentStep = #JOB_20_STEP_30) AND "Unit1.Em5.ControlNodes".gaugeRnR.sequence.status.seqActive AND "Unit1.Em5.ControlNodes".gaugeRnR."step".transition1[2030] THEN
       "Unit1.Em5.ControlNodes".gaugeRnR.sequence.status.nextStep := #JOB_20_STEP_40;
   END_IF;
END_REGION

REGION Network 98: Step[2040] : MainPnP2 Z-axis Up
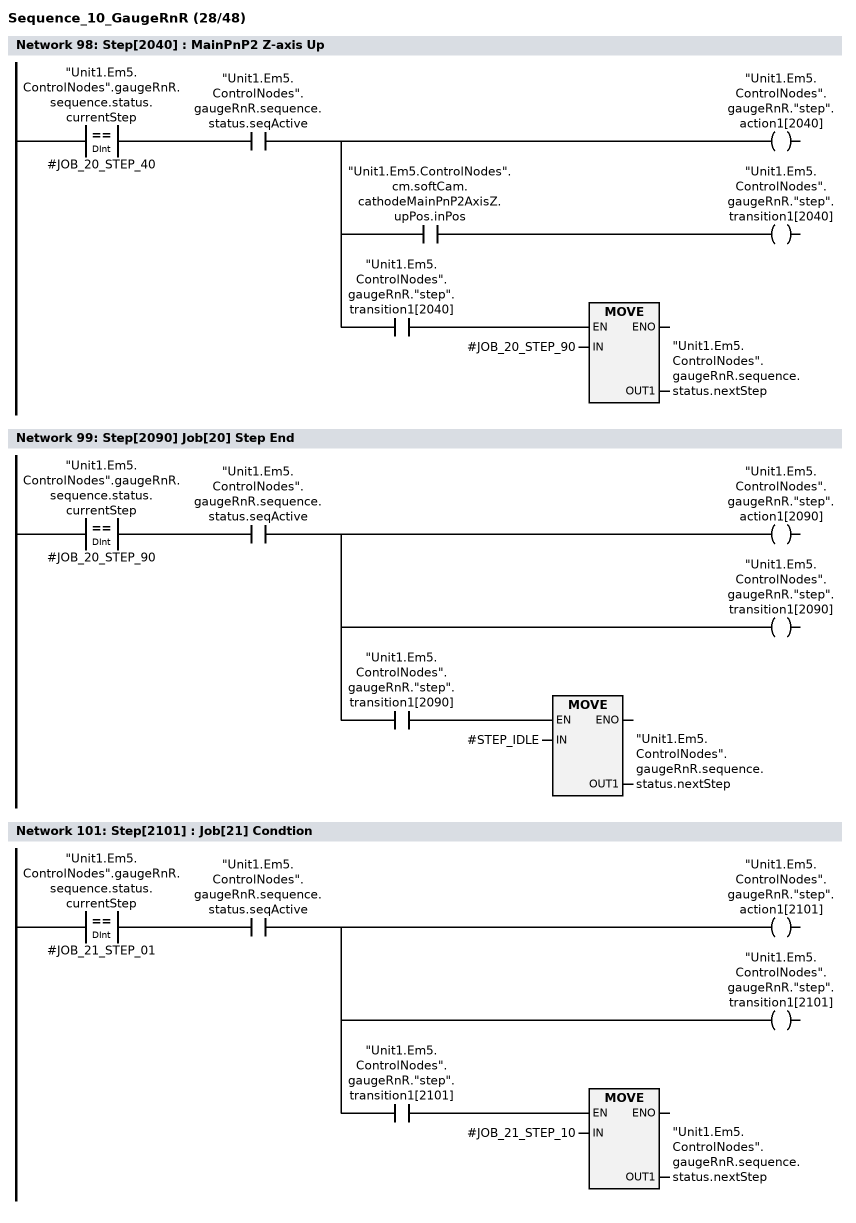
   RUNG wire#powerrail
      { S7_Templates := "SrcType := DInt" } EQ_Contact(in1 := "Unit1.Em5.ControlNodes".gaugeRnR.sequence.status.currentStep, in2 := #JOB_20_STEP_40)
      Contact( "Unit1.Em5.ControlNodes".gaugeRnR.sequence.status.seqActive )
      wire#w1
      Coil( "Unit1.Em5.ControlNodes".gaugeRnR."step".action1[2040] )
   END_RUNG
   RUNG wire#w1
      Contact( "Unit1.Em5.ControlNodes".cm.softCam.cathodeMainPnP2AxisZ.upPos.inPos )
      Coil( "Unit1.Em5.ControlNodes".gaugeRnR."step".transition1[2040] )
   END_RUNG
   RUNG wire#w1
      Contact( "Unit1.Em5.ControlNodes".gaugeRnR."step".transition1[2040] )
      Move(in := #JOB_20_STEP_90, out1 => "Unit1.Em5.ControlNodes".gaugeRnR.sequence.status.nextStep)
   END_RUNG
   // the same network as SCL:
   "Unit1.Em5.ControlNodes".gaugeRnR."step".action1[2040] := ("Unit1.Em5.ControlNodes".gaugeRnR.sequence.status.currentStep = #JOB_20_STEP_40) AND "Unit1.Em5.ControlNodes".gaugeRnR.sequence.status.seqActive;
   "Unit1.Em5.ControlNodes".gaugeRnR."step".transition1[2040] := ("Unit1.Em5.ControlNodes".gaugeRnR.sequence.status.currentStep = #JOB_20_STEP_40) AND "Unit1.Em5.ControlNodes".gaugeRnR.sequence.status.seqActive AND "Unit1.Em5.ControlNodes".cm.softCam.cathodeMainPnP2AxisZ.upPos.inPos;
   IF ("Unit1.Em5.ControlNodes".gaugeRnR.sequence.status.currentStep = #JOB_20_STEP_40) AND "Unit1.Em5.ControlNodes".gaugeRnR.sequence.status.seqActive AND "Unit1.Em5.ControlNodes".gaugeRnR."step".transition1[2040] THEN
       "Unit1.Em5.ControlNodes".gaugeRnR.sequence.status.nextStep := #JOB_20_STEP_90;
   END_IF;
END_REGION

REGION Network 99: Step[2090] Job[20] Step End
   RUNG wire#powerrail
      { S7_Templates := "SrcType := DInt" } EQ_Contact(in1 := "Unit1.Em5.ControlNodes".gaugeRnR.sequence.status.currentStep, in2 := #JOB_20_STEP_90)
      Contact( "Unit1.Em5.ControlNodes".gaugeRnR.sequence.status.seqActive )
      wire#w1
      Coil( "Unit1.Em5.ControlNodes".gaugeRnR."step".action1[2090] )
   END_RUNG
   RUNG wire#w1
      Coil( "Unit1.Em5.ControlNodes".gaugeRnR."step".transition1[2090] )
   END_RUNG
   RUNG wire#w1
      Contact( "Unit1.Em5.ControlNodes".gaugeRnR."step".transition1[2090] )
      Move(in := #STEP_IDLE, out1 => "Unit1.Em5.ControlNodes".gaugeRnR.sequence.status.nextStep)
   END_RUNG
   // the same network as SCL:
   "Unit1.Em5.ControlNodes".gaugeRnR."step".action1[2090] := ("Unit1.Em5.ControlNodes".gaugeRnR.sequence.status.currentStep = #JOB_20_STEP_90) AND "Unit1.Em5.ControlNodes".gaugeRnR.sequence.status.seqActive;
   "Unit1.Em5.ControlNodes".gaugeRnR."step".transition1[2090] := ("Unit1.Em5.ControlNodes".gaugeRnR.sequence.status.currentStep = #JOB_20_STEP_90) AND "Unit1.Em5.ControlNodes".gaugeRnR.sequence.status.seqActive;
   IF ("Unit1.Em5.ControlNodes".gaugeRnR.sequence.status.currentStep = #JOB_20_STEP_90) AND "Unit1.Em5.ControlNodes".gaugeRnR.sequence.status.seqActive AND "Unit1.Em5.ControlNodes".gaugeRnR."step".transition1[2090] THEN
       "Unit1.Em5.ControlNodes".gaugeRnR.sequence.status.nextStep := #STEP_IDLE;
   END_IF;
END_REGION

REGION Network 100: *************** JOB[21] MainPnP Move ReelCut Convyeor / AlignTable************************
END_REGION

REGION Network 101: Step[2101] : Job[21] Condtion
   RUNG wire#powerrail
      { S7_Templates := "SrcType := DInt" } EQ_Contact(in1 := "Unit1.Em5.ControlNodes".gaugeRnR.sequence.status.currentStep, in2 := #JOB_21_STEP_01)
      Contact( "Unit1.Em5.ControlNodes".gaugeRnR.sequence.status.seqActive )
      wire#w1
      Coil( "Unit1.Em5.ControlNodes".gaugeRnR."step".action1[2101] )
   END_RUNG
   RUNG wire#w1
      Coil( "Unit1.Em5.ControlNodes".gaugeRnR."step".transition1[2101] )
   END_RUNG
   RUNG wire#w1
      Contact( "Unit1.Em5.ControlNodes".gaugeRnR."step".transition1[2101] )
      Move(in := #JOB_21_STEP_10, out1 => "Unit1.Em5.ControlNodes".gaugeRnR.sequence.status.nextStep)
   END_RUNG
   // the same network as SCL:
   "Unit1.Em5.ControlNodes".gaugeRnR."step".action1[2101] := ("Unit1.Em5.ControlNodes".gaugeRnR.sequence.status.currentStep = #JOB_21_STEP_01) AND "Unit1.Em5.ControlNodes".gaugeRnR.sequence.status.seqActive;
   "Unit1.Em5.ControlNodes".gaugeRnR."step".transition1[2101] := ("Unit1.Em5.ControlNodes".gaugeRnR.sequence.status.currentStep = #JOB_21_STEP_01) AND "Unit1.Em5.ControlNodes".gaugeRnR.sequence.status.seqActive;
   IF ("Unit1.Em5.ControlNodes".gaugeRnR.sequence.status.currentStep = #JOB_21_STEP_01) AND "Unit1.Em5.ControlNodes".gaugeRnR.sequence.status.seqActive AND "Unit1.Em5.ControlNodes".gaugeRnR."step".transition1[2101] THEN
       "Unit1.Em5.ControlNodes".gaugeRnR.sequence.status.nextStep := #JOB_21_STEP_10;
   END_IF;
END_REGION

REGION Network 102: Step[2110] : MainPnP1 X-Axis Move ReelCut Convyeor
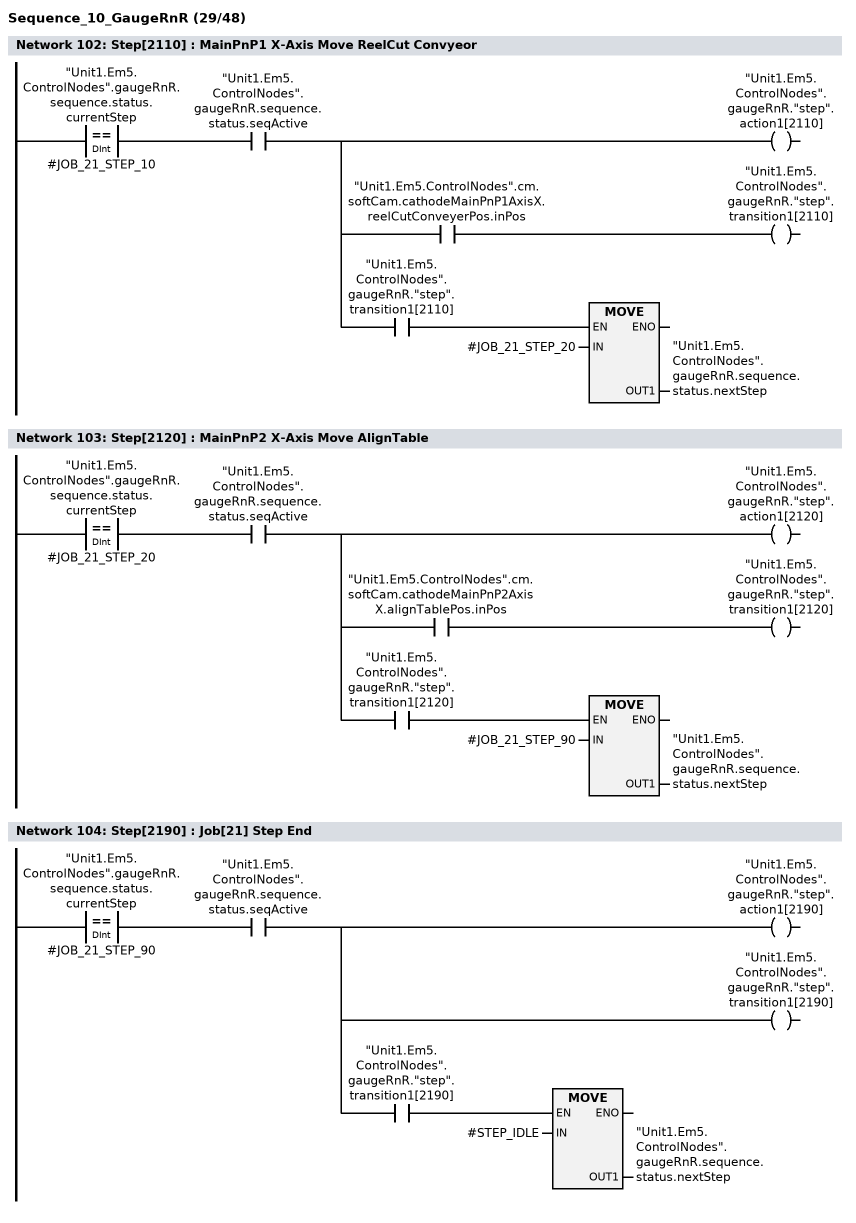
   RUNG wire#powerrail
      { S7_Templates := "SrcType := DInt" } EQ_Contact(in1 := "Unit1.Em5.ControlNodes".gaugeRnR.sequence.status.currentStep, in2 := #JOB_21_STEP_10)
      Contact( "Unit1.Em5.ControlNodes".gaugeRnR.sequence.status.seqActive )
      wire#w1
      Coil( "Unit1.Em5.ControlNodes".gaugeRnR."step".action1[2110] )
   END_RUNG
   RUNG wire#w1
      Contact( "Unit1.Em5.ControlNodes".cm.softCam.cathodeMainPnP1AxisX.reelCutConveyerPos.inPos )
      Coil( "Unit1.Em5.ControlNodes".gaugeRnR."step".transition1[2110] )
   END_RUNG
   RUNG wire#w1
      Contact( "Unit1.Em5.ControlNodes".gaugeRnR."step".transition1[2110] )
      Move(in := #JOB_21_STEP_20, out1 => "Unit1.Em5.ControlNodes".gaugeRnR.sequence.status.nextStep)
   END_RUNG
   // the same network as SCL:
   "Unit1.Em5.ControlNodes".gaugeRnR."step".action1[2110] := ("Unit1.Em5.ControlNodes".gaugeRnR.sequence.status.currentStep = #JOB_21_STEP_10) AND "Unit1.Em5.ControlNodes".gaugeRnR.sequence.status.seqActive;
   "Unit1.Em5.ControlNodes".gaugeRnR."step".transition1[2110] := ("Unit1.Em5.ControlNodes".gaugeRnR.sequence.status.currentStep = #JOB_21_STEP_10) AND "Unit1.Em5.ControlNodes".gaugeRnR.sequence.status.seqActive AND "Unit1.Em5.ControlNodes".cm.softCam.cathodeMainPnP1AxisX.reelCutConveyerPos.inPos;
   IF ("Unit1.Em5.ControlNodes".gaugeRnR.sequence.status.currentStep = #JOB_21_STEP_10) AND "Unit1.Em5.ControlNodes".gaugeRnR.sequence.status.seqActive AND "Unit1.Em5.ControlNodes".gaugeRnR."step".transition1[2110] THEN
       "Unit1.Em5.ControlNodes".gaugeRnR.sequence.status.nextStep := #JOB_21_STEP_20;
   END_IF;
END_REGION

REGION Network 103: Step[2120] : MainPnP2 X-Axis Move AlignTable
   RUNG wire#powerrail
      { S7_Templates := "SrcType := DInt" } EQ_Contact(in1 := "Unit1.Em5.ControlNodes".gaugeRnR.sequence.status.currentStep, in2 := #JOB_21_STEP_20)
      Contact( "Unit1.Em5.ControlNodes".gaugeRnR.sequence.status.seqActive )
      wire#w1
      Coil( "Unit1.Em5.ControlNodes".gaugeRnR."step".action1[2120] )
   END_RUNG
   RUNG wire#w1
      Contact( "Unit1.Em5.ControlNodes".cm.softCam.cathodeMainPnP2AxisX.alignTablePos.inPos )
      Coil( "Unit1.Em5.ControlNodes".gaugeRnR."step".transition1[2120] )
   END_RUNG
   RUNG wire#w1
      Contact( "Unit1.Em5.ControlNodes".gaugeRnR."step".transition1[2120] )
      Move(in := #JOB_21_STEP_90, out1 => "Unit1.Em5.ControlNodes".gaugeRnR.sequence.status.nextStep)
   END_RUNG
   // the same network as SCL:
   "Unit1.Em5.ControlNodes".gaugeRnR."step".action1[2120] := ("Unit1.Em5.ControlNodes".gaugeRnR.sequence.status.currentStep = #JOB_21_STEP_20) AND "Unit1.Em5.ControlNodes".gaugeRnR.sequence.status.seqActive;
   "Unit1.Em5.ControlNodes".gaugeRnR."step".transition1[2120] := ("Unit1.Em5.ControlNodes".gaugeRnR.sequence.status.currentStep = #JOB_21_STEP_20) AND "Unit1.Em5.ControlNodes".gaugeRnR.sequence.status.seqActive AND "Unit1.Em5.ControlNodes".cm.softCam.cathodeMainPnP2AxisX.alignTablePos.inPos;
   IF ("Unit1.Em5.ControlNodes".gaugeRnR.sequence.status.currentStep = #JOB_21_STEP_20) AND "Unit1.Em5.ControlNodes".gaugeRnR.sequence.status.seqActive AND "Unit1.Em5.ControlNodes".gaugeRnR."step".transition1[2120] THEN
       "Unit1.Em5.ControlNodes".gaugeRnR.sequence.status.nextStep := #JOB_21_STEP_90;
   END_IF;
END_REGION

REGION Network 104: Step[2190] : Job[21] Step End
   RUNG wire#powerrail
      { S7_Templates := "SrcType := DInt" } EQ_Contact(in1 := "Unit1.Em5.ControlNodes".gaugeRnR.sequence.status.currentStep, in2 := #JOB_21_STEP_90)
      Contact( "Unit1.Em5.ControlNodes".gaugeRnR.sequence.status.seqActive )
      wire#w1
      Coil( "Unit1.Em5.ControlNodes".gaugeRnR."step".action1[2190] )
   END_RUNG
   RUNG wire#w1
      Coil( "Unit1.Em5.ControlNodes".gaugeRnR."step".transition1[2190] )
   END_RUNG
   RUNG wire#w1
      Contact( "Unit1.Em5.ControlNodes".gaugeRnR."step".transition1[2190] )
      Move(in := #STEP_IDLE, out1 => "Unit1.Em5.ControlNodes".gaugeRnR.sequence.status.nextStep)
   END_RUNG
   // the same network as SCL:
   "Unit1.Em5.ControlNodes".gaugeRnR."step".action1[2190] := ("Unit1.Em5.ControlNodes".gaugeRnR.sequence.status.currentStep = #JOB_21_STEP_90) AND "Unit1.Em5.ControlNodes".gaugeRnR.sequence.status.seqActive;
   "Unit1.Em5.ControlNodes".gaugeRnR."step".transition1[2190] := ("Unit1.Em5.ControlNodes".gaugeRnR.sequence.status.currentStep = #JOB_21_STEP_90) AND "Unit1.Em5.ControlNodes".gaugeRnR.sequence.status.seqActive;
   IF ("Unit1.Em5.ControlNodes".gaugeRnR.sequence.status.currentStep = #JOB_21_STEP_90) AND "Unit1.Em5.ControlNodes".gaugeRnR.sequence.status.seqActive AND "Unit1.Em5.ControlNodes".gaugeRnR."step".transition1[2190] THEN
       "Unit1.Em5.ControlNodes".gaugeRnR.sequence.status.nextStep := #STEP_IDLE;
   END_IF;
END_REGION

REGION Network 105: *************** JOB[22] MainPnP2 To AlignTable ************************
END_REGION

REGION Network 106: Step[2201] : Job[22] Condtion
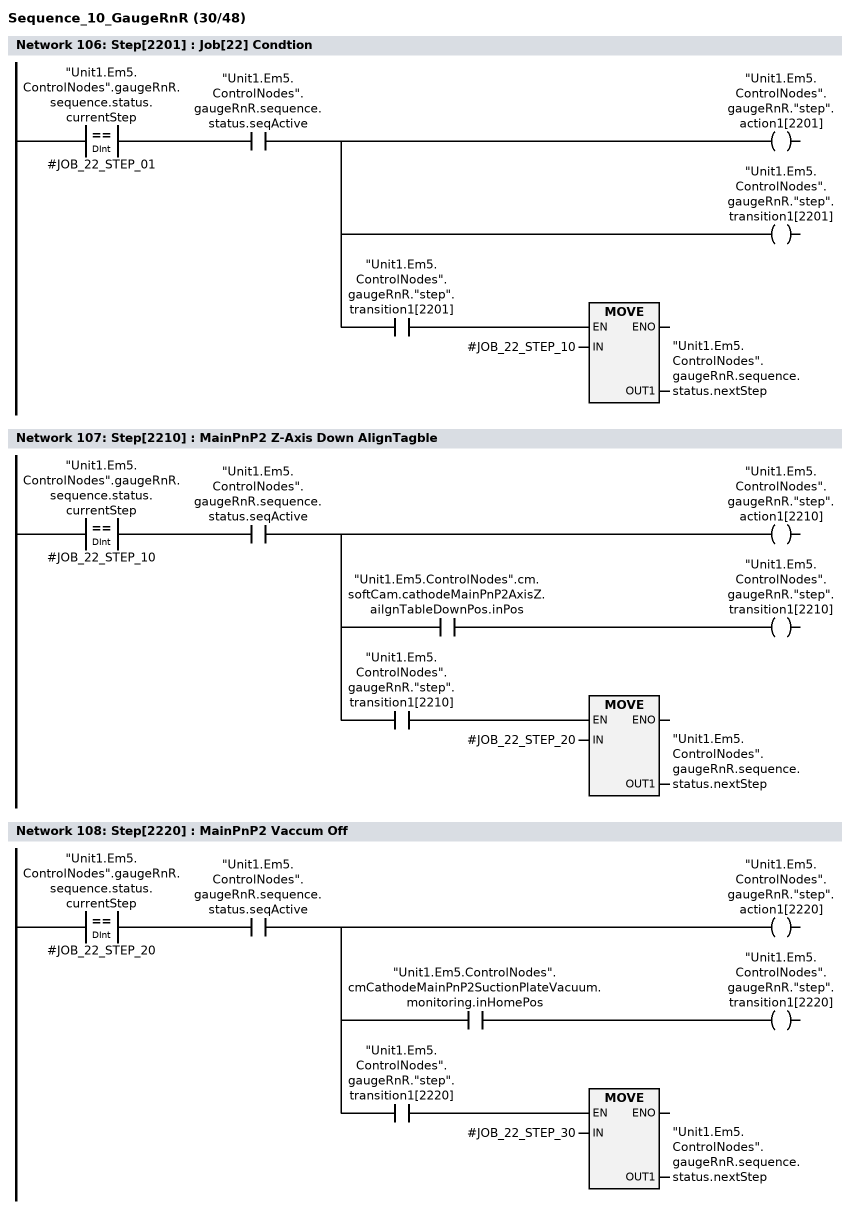
   RUNG wire#powerrail
      { S7_Templates := "SrcType := DInt" } EQ_Contact(in1 := "Unit1.Em5.ControlNodes".gaugeRnR.sequence.status.currentStep, in2 := #JOB_22_STEP_01)
      Contact( "Unit1.Em5.ControlNodes".gaugeRnR.sequence.status.seqActive )
      wire#w1
      Coil( "Unit1.Em5.ControlNodes".gaugeRnR."step".action1[2201] )
   END_RUNG
   RUNG wire#w1
      Coil( "Unit1.Em5.ControlNodes".gaugeRnR."step".transition1[2201] )
   END_RUNG
   RUNG wire#w1
      Contact( "Unit1.Em5.ControlNodes".gaugeRnR."step".transition1[2201] )
      Move(in := #JOB_22_STEP_10, out1 => "Unit1.Em5.ControlNodes".gaugeRnR.sequence.status.nextStep)
   END_RUNG
   // the same network as SCL:
   "Unit1.Em5.ControlNodes".gaugeRnR."step".action1[2201] := ("Unit1.Em5.ControlNodes".gaugeRnR.sequence.status.currentStep = #JOB_22_STEP_01) AND "Unit1.Em5.ControlNodes".gaugeRnR.sequence.status.seqActive;
   "Unit1.Em5.ControlNodes".gaugeRnR."step".transition1[2201] := ("Unit1.Em5.ControlNodes".gaugeRnR.sequence.status.currentStep = #JOB_22_STEP_01) AND "Unit1.Em5.ControlNodes".gaugeRnR.sequence.status.seqActive;
   IF ("Unit1.Em5.ControlNodes".gaugeRnR.sequence.status.currentStep = #JOB_22_STEP_01) AND "Unit1.Em5.ControlNodes".gaugeRnR.sequence.status.seqActive AND "Unit1.Em5.ControlNodes".gaugeRnR."step".transition1[2201] THEN
       "Unit1.Em5.ControlNodes".gaugeRnR.sequence.status.nextStep := #JOB_22_STEP_10;
   END_IF;
END_REGION

REGION Network 107: Step[2210] : MainPnP2 Z-Axis Down AlignTagble
   RUNG wire#powerrail
      { S7_Templates := "SrcType := DInt" } EQ_Contact(in1 := "Unit1.Em5.ControlNodes".gaugeRnR.sequence.status.currentStep, in2 := #JOB_22_STEP_10)
      Contact( "Unit1.Em5.ControlNodes".gaugeRnR.sequence.status.seqActive )
      wire#w1
      Coil( "Unit1.Em5.ControlNodes".gaugeRnR."step".action1[2210] )
   END_RUNG
   RUNG wire#w1
      Contact( "Unit1.Em5.ControlNodes".cm.softCam.cathodeMainPnP2AxisZ.ailgnTableDownPos.inPos )
      Coil( "Unit1.Em5.ControlNodes".gaugeRnR."step".transition1[2210] )
   END_RUNG
   RUNG wire#w1
      Contact( "Unit1.Em5.ControlNodes".gaugeRnR."step".transition1[2210] )
      Move(in := #JOB_22_STEP_20, out1 => "Unit1.Em5.ControlNodes".gaugeRnR.sequence.status.nextStep)
   END_RUNG
   // the same network as SCL:
   "Unit1.Em5.ControlNodes".gaugeRnR."step".action1[2210] := ("Unit1.Em5.ControlNodes".gaugeRnR.sequence.status.currentStep = #JOB_22_STEP_10) AND "Unit1.Em5.ControlNodes".gaugeRnR.sequence.status.seqActive;
   "Unit1.Em5.ControlNodes".gaugeRnR."step".transition1[2210] := ("Unit1.Em5.ControlNodes".gaugeRnR.sequence.status.currentStep = #JOB_22_STEP_10) AND "Unit1.Em5.ControlNodes".gaugeRnR.sequence.status.seqActive AND "Unit1.Em5.ControlNodes".cm.softCam.cathodeMainPnP2AxisZ.ailgnTableDownPos.inPos;
   IF ("Unit1.Em5.ControlNodes".gaugeRnR.sequence.status.currentStep = #JOB_22_STEP_10) AND "Unit1.Em5.ControlNodes".gaugeRnR.sequence.status.seqActive AND "Unit1.Em5.ControlNodes".gaugeRnR."step".transition1[2210] THEN
       "Unit1.Em5.ControlNodes".gaugeRnR.sequence.status.nextStep := #JOB_22_STEP_20;
   END_IF;
END_REGION

REGION Network 108: Step[2220] : MainPnP2 Vaccum Off
   RUNG wire#powerrail
      { S7_Templates := "SrcType := DInt" } EQ_Contact(in1 := "Unit1.Em5.ControlNodes".gaugeRnR.sequence.status.currentStep, in2 := #JOB_22_STEP_20)
      Contact( "Unit1.Em5.ControlNodes".gaugeRnR.sequence.status.seqActive )
      wire#w1
      Coil( "Unit1.Em5.ControlNodes".gaugeRnR."step".action1[2220] )
   END_RUNG
   RUNG wire#w1
      Contact( "Unit1.Em5.ControlNodes".cmCathodeMainPnP2SuctionPlateVacuum.monitoring.inHomePos )
      Coil( "Unit1.Em5.ControlNodes".gaugeRnR."step".transition1[2220] )
   END_RUNG
   RUNG wire#w1
      Contact( "Unit1.Em5.ControlNodes".gaugeRnR."step".transition1[2220] )
      Move(in := #JOB_22_STEP_30, out1 => "Unit1.Em5.ControlNodes".gaugeRnR.sequence.status.nextStep)
   END_RUNG
   // the same network as SCL:
   "Unit1.Em5.ControlNodes".gaugeRnR."step".action1[2220] := ("Unit1.Em5.ControlNodes".gaugeRnR.sequence.status.currentStep = #JOB_22_STEP_20) AND "Unit1.Em5.ControlNodes".gaugeRnR.sequence.status.seqActive;
   "Unit1.Em5.ControlNodes".gaugeRnR."step".transition1[2220] := ("Unit1.Em5.ControlNodes".gaugeRnR.sequence.status.currentStep = #JOB_22_STEP_20) AND "Unit1.Em5.ControlNodes".gaugeRnR.sequence.status.seqActive AND "Unit1.Em5.ControlNodes".cmCathodeMainPnP2SuctionPlateVacuum.monitoring.inHomePos;
   IF ("Unit1.Em5.ControlNodes".gaugeRnR.sequence.status.currentStep = #JOB_22_STEP_20) AND "Unit1.Em5.ControlNodes".gaugeRnR.sequence.status.seqActive AND "Unit1.Em5.ControlNodes".gaugeRnR."step".transition1[2220] THEN
       "Unit1.Em5.ControlNodes".gaugeRnR.sequence.status.nextStep := #JOB_22_STEP_30;
   END_IF;
END_REGION

REGION Network 109: Step[2230] : AlignTable Vaccum On
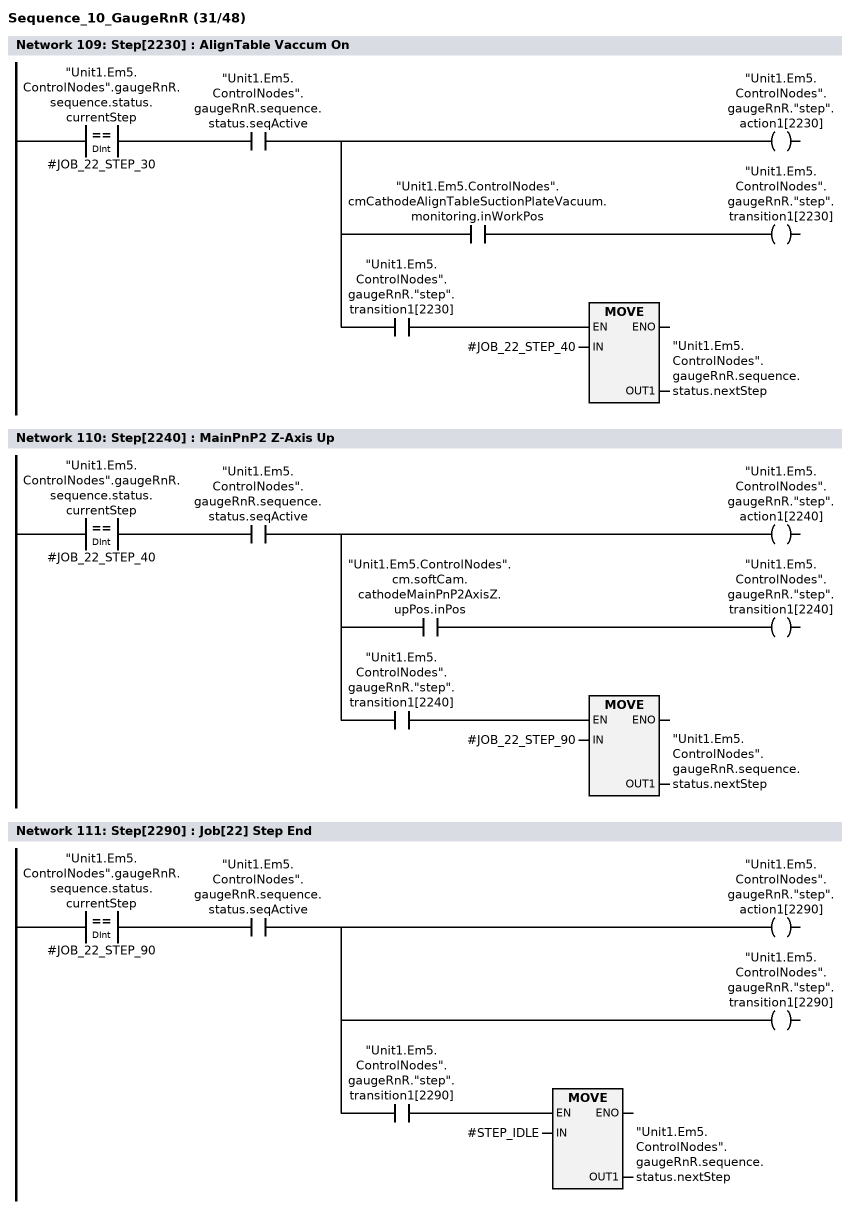
   RUNG wire#powerrail
      { S7_Templates := "SrcType := DInt" } EQ_Contact(in1 := "Unit1.Em5.ControlNodes".gaugeRnR.sequence.status.currentStep, in2 := #JOB_22_STEP_30)
      Contact( "Unit1.Em5.ControlNodes".gaugeRnR.sequence.status.seqActive )
      wire#w1
      Coil( "Unit1.Em5.ControlNodes".gaugeRnR."step".action1[2230] )
   END_RUNG
   RUNG wire#w1
      Contact( "Unit1.Em5.ControlNodes".cmCathodeAlignTableSuctionPlateVacuum.monitoring.inWorkPos )
      Coil( "Unit1.Em5.ControlNodes".gaugeRnR."step".transition1[2230] )
   END_RUNG
   RUNG wire#w1
      Contact( "Unit1.Em5.ControlNodes".gaugeRnR."step".transition1[2230] )
      Move(in := #JOB_22_STEP_40, out1 => "Unit1.Em5.ControlNodes".gaugeRnR.sequence.status.nextStep)
   END_RUNG
   // the same network as SCL:
   "Unit1.Em5.ControlNodes".gaugeRnR."step".action1[2230] := ("Unit1.Em5.ControlNodes".gaugeRnR.sequence.status.currentStep = #JOB_22_STEP_30) AND "Unit1.Em5.ControlNodes".gaugeRnR.sequence.status.seqActive;
   "Unit1.Em5.ControlNodes".gaugeRnR."step".transition1[2230] := ("Unit1.Em5.ControlNodes".gaugeRnR.sequence.status.currentStep = #JOB_22_STEP_30) AND "Unit1.Em5.ControlNodes".gaugeRnR.sequence.status.seqActive AND "Unit1.Em5.ControlNodes".cmCathodeAlignTableSuctionPlateVacuum.monitoring.inWorkPos;
   IF ("Unit1.Em5.ControlNodes".gaugeRnR.sequence.status.currentStep = #JOB_22_STEP_30) AND "Unit1.Em5.ControlNodes".gaugeRnR.sequence.status.seqActive AND "Unit1.Em5.ControlNodes".gaugeRnR."step".transition1[2230] THEN
       "Unit1.Em5.ControlNodes".gaugeRnR.sequence.status.nextStep := #JOB_22_STEP_40;
   END_IF;
END_REGION

REGION Network 110: Step[2240] : MainPnP2 Z-Axis Up
   RUNG wire#powerrail
      { S7_Templates := "SrcType := DInt" } EQ_Contact(in1 := "Unit1.Em5.ControlNodes".gaugeRnR.sequence.status.currentStep, in2 := #JOB_22_STEP_40)
      Contact( "Unit1.Em5.ControlNodes".gaugeRnR.sequence.status.seqActive )
      wire#w1
      Coil( "Unit1.Em5.ControlNodes".gaugeRnR."step".action1[2240] )
   END_RUNG
   RUNG wire#w1
      Contact( "Unit1.Em5.ControlNodes".cm.softCam.cathodeMainPnP2AxisZ.upPos.inPos )
      Coil( "Unit1.Em5.ControlNodes".gaugeRnR."step".transition1[2240] )
   END_RUNG
   RUNG wire#w1
      Contact( "Unit1.Em5.ControlNodes".gaugeRnR."step".transition1[2240] )
      Move(in := #JOB_22_STEP_90, out1 => "Unit1.Em5.ControlNodes".gaugeRnR.sequence.status.nextStep)
   END_RUNG
   // the same network as SCL:
   "Unit1.Em5.ControlNodes".gaugeRnR."step".action1[2240] := ("Unit1.Em5.ControlNodes".gaugeRnR.sequence.status.currentStep = #JOB_22_STEP_40) AND "Unit1.Em5.ControlNodes".gaugeRnR.sequence.status.seqActive;
   "Unit1.Em5.ControlNodes".gaugeRnR."step".transition1[2240] := ("Unit1.Em5.ControlNodes".gaugeRnR.sequence.status.currentStep = #JOB_22_STEP_40) AND "Unit1.Em5.ControlNodes".gaugeRnR.sequence.status.seqActive AND "Unit1.Em5.ControlNodes".cm.softCam.cathodeMainPnP2AxisZ.upPos.inPos;
   IF ("Unit1.Em5.ControlNodes".gaugeRnR.sequence.status.currentStep = #JOB_22_STEP_40) AND "Unit1.Em5.ControlNodes".gaugeRnR.sequence.status.seqActive AND "Unit1.Em5.ControlNodes".gaugeRnR."step".transition1[2240] THEN
       "Unit1.Em5.ControlNodes".gaugeRnR.sequence.status.nextStep := #JOB_22_STEP_90;
   END_IF;
END_REGION

REGION Network 111: Step[2290] : Job[22] Step End
   RUNG wire#powerrail
      { S7_Templates := "SrcType := DInt" } EQ_Contact(in1 := "Unit1.Em5.ControlNodes".gaugeRnR.sequence.status.currentStep, in2 := #JOB_22_STEP_90)
      Contact( "Unit1.Em5.ControlNodes".gaugeRnR.sequence.status.seqActive )
      wire#w1
      Coil( "Unit1.Em5.ControlNodes".gaugeRnR."step".action1[2290] )
   END_RUNG
   RUNG wire#w1
      Coil( "Unit1.Em5.ControlNodes".gaugeRnR."step".transition1[2290] )
   END_RUNG
   RUNG wire#w1
      Contact( "Unit1.Em5.ControlNodes".gaugeRnR."step".transition1[2290] )
      Move(in := #STEP_IDLE, out1 => "Unit1.Em5.ControlNodes".gaugeRnR.sequence.status.nextStep)
   END_RUNG
   // the same network as SCL:
   "Unit1.Em5.ControlNodes".gaugeRnR."step".action1[2290] := ("Unit1.Em5.ControlNodes".gaugeRnR.sequence.status.currentStep = #JOB_22_STEP_90) AND "Unit1.Em5.ControlNodes".gaugeRnR.sequence.status.seqActive;
   "Unit1.Em5.ControlNodes".gaugeRnR."step".transition1[2290] := ("Unit1.Em5.ControlNodes".gaugeRnR.sequence.status.currentStep = #JOB_22_STEP_90) AND "Unit1.Em5.ControlNodes".gaugeRnR.sequence.status.seqActive;
   IF ("Unit1.Em5.ControlNodes".gaugeRnR.sequence.status.currentStep = #JOB_22_STEP_90) AND "Unit1.Em5.ControlNodes".gaugeRnR.sequence.status.seqActive AND "Unit1.Em5.ControlNodes".gaugeRnR."step".transition1[2290] THEN
       "Unit1.Em5.ControlNodes".gaugeRnR.sequence.status.nextStep := #STEP_IDLE;
   END_IF;
END_REGION

REGION Network 112: *************** JOB[23] MainPnP Move AlignTable / StackTable ************************
END_REGION

REGION Network 113: Step[2301] : JOB[23] Condition
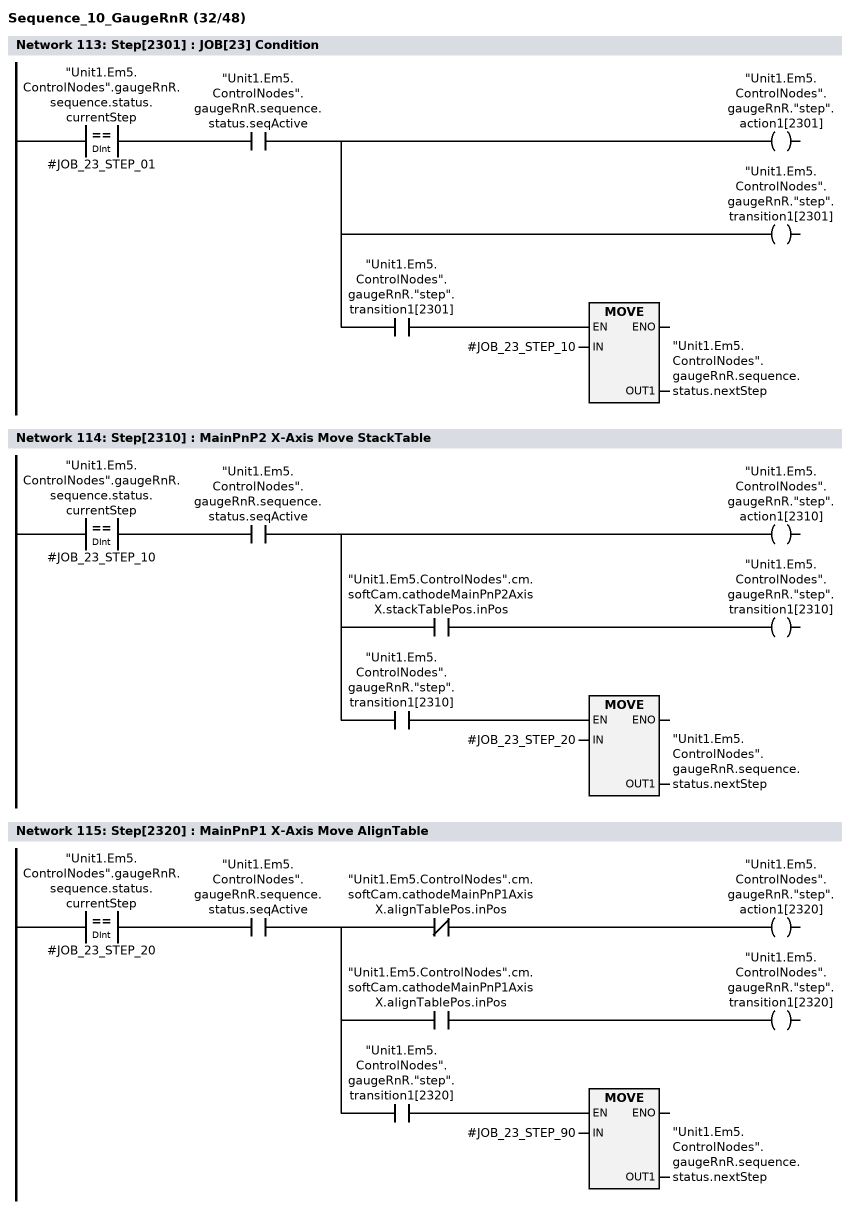
   RUNG wire#powerrail
      { S7_Templates := "SrcType := DInt" } EQ_Contact(in1 := "Unit1.Em5.ControlNodes".gaugeRnR.sequence.status.currentStep, in2 := #JOB_23_STEP_01)
      Contact( "Unit1.Em5.ControlNodes".gaugeRnR.sequence.status.seqActive )
      wire#w1
      Coil( "Unit1.Em5.ControlNodes".gaugeRnR."step".action1[2301] )
   END_RUNG
   RUNG wire#w1
      Coil( "Unit1.Em5.ControlNodes".gaugeRnR."step".transition1[2301] )
   END_RUNG
   RUNG wire#w1
      Contact( "Unit1.Em5.ControlNodes".gaugeRnR."step".transition1[2301] )
      Move(in := #JOB_23_STEP_10, out1 => "Unit1.Em5.ControlNodes".gaugeRnR.sequence.status.nextStep)
   END_RUNG
   // the same network as SCL:
   "Unit1.Em5.ControlNodes".gaugeRnR."step".action1[2301] := ("Unit1.Em5.ControlNodes".gaugeRnR.sequence.status.currentStep = #JOB_23_STEP_01) AND "Unit1.Em5.ControlNodes".gaugeRnR.sequence.status.seqActive;
   "Unit1.Em5.ControlNodes".gaugeRnR."step".transition1[2301] := ("Unit1.Em5.ControlNodes".gaugeRnR.sequence.status.currentStep = #JOB_23_STEP_01) AND "Unit1.Em5.ControlNodes".gaugeRnR.sequence.status.seqActive;
   IF ("Unit1.Em5.ControlNodes".gaugeRnR.sequence.status.currentStep = #JOB_23_STEP_01) AND "Unit1.Em5.ControlNodes".gaugeRnR.sequence.status.seqActive AND "Unit1.Em5.ControlNodes".gaugeRnR."step".transition1[2301] THEN
       "Unit1.Em5.ControlNodes".gaugeRnR.sequence.status.nextStep := #JOB_23_STEP_10;
   END_IF;
END_REGION

REGION Network 114: Step[2310] : MainPnP2 X-Axis Move StackTable
   RUNG wire#powerrail
      { S7_Templates := "SrcType := DInt" } EQ_Contact(in1 := "Unit1.Em5.ControlNodes".gaugeRnR.sequence.status.currentStep, in2 := #JOB_23_STEP_10)
      Contact( "Unit1.Em5.ControlNodes".gaugeRnR.sequence.status.seqActive )
      wire#w1
      Coil( "Unit1.Em5.ControlNodes".gaugeRnR."step".action1[2310] )
   END_RUNG
   RUNG wire#w1
      Contact( "Unit1.Em5.ControlNodes".cm.softCam.cathodeMainPnP2AxisX.stackTablePos.inPos )
      Coil( "Unit1.Em5.ControlNodes".gaugeRnR."step".transition1[2310] )
   END_RUNG
   RUNG wire#w1
      Contact( "Unit1.Em5.ControlNodes".gaugeRnR."step".transition1[2310] )
      Move(in := #JOB_23_STEP_20, out1 => "Unit1.Em5.ControlNodes".gaugeRnR.sequence.status.nextStep)
   END_RUNG
   // the same network as SCL:
   "Unit1.Em5.ControlNodes".gaugeRnR."step".action1[2310] := ("Unit1.Em5.ControlNodes".gaugeRnR.sequence.status.currentStep = #JOB_23_STEP_10) AND "Unit1.Em5.ControlNodes".gaugeRnR.sequence.status.seqActive;
   "Unit1.Em5.ControlNodes".gaugeRnR."step".transition1[2310] := ("Unit1.Em5.ControlNodes".gaugeRnR.sequence.status.currentStep = #JOB_23_STEP_10) AND "Unit1.Em5.ControlNodes".gaugeRnR.sequence.status.seqActive AND "Unit1.Em5.ControlNodes".cm.softCam.cathodeMainPnP2AxisX.stackTablePos.inPos;
   IF ("Unit1.Em5.ControlNodes".gaugeRnR.sequence.status.currentStep = #JOB_23_STEP_10) AND "Unit1.Em5.ControlNodes".gaugeRnR.sequence.status.seqActive AND "Unit1.Em5.ControlNodes".gaugeRnR."step".transition1[2310] THEN
       "Unit1.Em5.ControlNodes".gaugeRnR.sequence.status.nextStep := #JOB_23_STEP_20;
   END_IF;
END_REGION

REGION Network 115: Step[2320] : MainPnP1 X-Axis Move AlignTable
   RUNG wire#powerrail
      { S7_Templates := "SrcType := DInt" } EQ_Contact(in1 := "Unit1.Em5.ControlNodes".gaugeRnR.sequence.status.currentStep, in2 := #JOB_23_STEP_20)
      Contact( "Unit1.Em5.ControlNodes".gaugeRnR.sequence.status.seqActive )
      wire#w1
      I_Contact( "Unit1.Em5.ControlNodes".cm.softCam.cathodeMainPnP1AxisX.alignTablePos.inPos )
      Coil( "Unit1.Em5.ControlNodes".gaugeRnR."step".action1[2320] )
   END_RUNG
   RUNG wire#w1
      Contact( "Unit1.Em5.ControlNodes".cm.softCam.cathodeMainPnP1AxisX.alignTablePos.inPos )
      Coil( "Unit1.Em5.ControlNodes".gaugeRnR."step".transition1[2320] )
   END_RUNG
   RUNG wire#w1
      Contact( "Unit1.Em5.ControlNodes".gaugeRnR."step".transition1[2320] )
      Move(in := #JOB_23_STEP_90, out1 => "Unit1.Em5.ControlNodes".gaugeRnR.sequence.status.nextStep)
   END_RUNG
   // the same network as SCL:
   #_w1 := ("Unit1.Em5.ControlNodes".gaugeRnR.sequence.status.currentStep = #JOB_23_STEP_20) AND "Unit1.Em5.ControlNodes".gaugeRnR.sequence.status.seqActive;
   "Unit1.Em5.ControlNodes".gaugeRnR."step".action1[2320] := #_w1 AND NOT "Unit1.Em5.ControlNodes".cm.softCam.cathodeMainPnP1AxisX.alignTablePos.inPos;
   "Unit1.Em5.ControlNodes".gaugeRnR."step".transition1[2320] := #_w1 AND "Unit1.Em5.ControlNodes".cm.softCam.cathodeMainPnP1AxisX.alignTablePos.inPos;
   IF #_w1 AND "Unit1.Em5.ControlNodes".gaugeRnR."step".transition1[2320] THEN
       "Unit1.Em5.ControlNodes".gaugeRnR.sequence.status.nextStep := #JOB_23_STEP_90;
   END_IF;
END_REGION

REGION Network 116: Step[2390] : Job[23] Step End
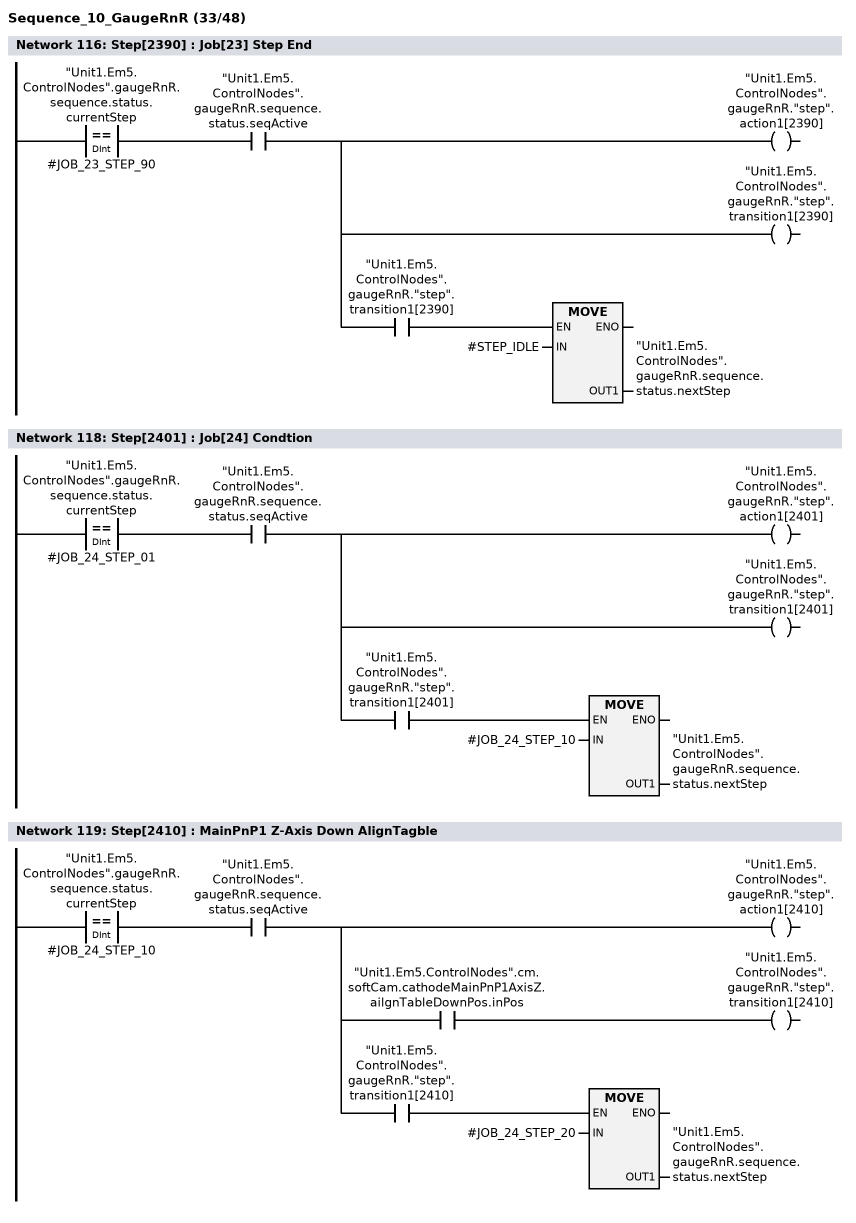
   RUNG wire#powerrail
      { S7_Templates := "SrcType := DInt" } EQ_Contact(in1 := "Unit1.Em5.ControlNodes".gaugeRnR.sequence.status.currentStep, in2 := #JOB_23_STEP_90)
      Contact( "Unit1.Em5.ControlNodes".gaugeRnR.sequence.status.seqActive )
      wire#w1
      Coil( "Unit1.Em5.ControlNodes".gaugeRnR."step".action1[2390] )
   END_RUNG
   RUNG wire#w1
      Coil( "Unit1.Em5.ControlNodes".gaugeRnR."step".transition1[2390] )
   END_RUNG
   RUNG wire#w1
      Contact( "Unit1.Em5.ControlNodes".gaugeRnR."step".transition1[2390] )
      Move(in := #STEP_IDLE, out1 => "Unit1.Em5.ControlNodes".gaugeRnR.sequence.status.nextStep)
   END_RUNG
   // the same network as SCL:
   "Unit1.Em5.ControlNodes".gaugeRnR."step".action1[2390] := ("Unit1.Em5.ControlNodes".gaugeRnR.sequence.status.currentStep = #JOB_23_STEP_90) AND "Unit1.Em5.ControlNodes".gaugeRnR.sequence.status.seqActive;
   "Unit1.Em5.ControlNodes".gaugeRnR."step".transition1[2390] := ("Unit1.Em5.ControlNodes".gaugeRnR.sequence.status.currentStep = #JOB_23_STEP_90) AND "Unit1.Em5.ControlNodes".gaugeRnR.sequence.status.seqActive;
   IF ("Unit1.Em5.ControlNodes".gaugeRnR.sequence.status.currentStep = #JOB_23_STEP_90) AND "Unit1.Em5.ControlNodes".gaugeRnR.sequence.status.seqActive AND "Unit1.Em5.ControlNodes".gaugeRnR."step".transition1[2390] THEN
       "Unit1.Em5.ControlNodes".gaugeRnR.sequence.status.nextStep := #STEP_IDLE;
   END_IF;
END_REGION

REGION Network 117: *************** JOB[24] AlignTable To MainPnP1 ************************
END_REGION

REGION Network 118: Step[2401] : Job[24] Condtion
   RUNG wire#powerrail
      { S7_Templates := "SrcType := DInt" } EQ_Contact(in1 := "Unit1.Em5.ControlNodes".gaugeRnR.sequence.status.currentStep, in2 := #JOB_24_STEP_01)
      Contact( "Unit1.Em5.ControlNodes".gaugeRnR.sequence.status.seqActive )
      wire#w1
      Coil( "Unit1.Em5.ControlNodes".gaugeRnR."step".action1[2401] )
   END_RUNG
   RUNG wire#w1
      Coil( "Unit1.Em5.ControlNodes".gaugeRnR."step".transition1[2401] )
   END_RUNG
   RUNG wire#w1
      Contact( "Unit1.Em5.ControlNodes".gaugeRnR."step".transition1[2401] )
      Move(in := #JOB_24_STEP_10, out1 => "Unit1.Em5.ControlNodes".gaugeRnR.sequence.status.nextStep)
   END_RUNG
   // the same network as SCL:
   "Unit1.Em5.ControlNodes".gaugeRnR."step".action1[2401] := ("Unit1.Em5.ControlNodes".gaugeRnR.sequence.status.currentStep = #JOB_24_STEP_01) AND "Unit1.Em5.ControlNodes".gaugeRnR.sequence.status.seqActive;
   "Unit1.Em5.ControlNodes".gaugeRnR."step".transition1[2401] := ("Unit1.Em5.ControlNodes".gaugeRnR.sequence.status.currentStep = #JOB_24_STEP_01) AND "Unit1.Em5.ControlNodes".gaugeRnR.sequence.status.seqActive;
   IF ("Unit1.Em5.ControlNodes".gaugeRnR.sequence.status.currentStep = #JOB_24_STEP_01) AND "Unit1.Em5.ControlNodes".gaugeRnR.sequence.status.seqActive AND "Unit1.Em5.ControlNodes".gaugeRnR."step".transition1[2401] THEN
       "Unit1.Em5.ControlNodes".gaugeRnR.sequence.status.nextStep := #JOB_24_STEP_10;
   END_IF;
END_REGION

REGION Network 119: Step[2410] : MainPnP1 Z-Axis Down AlignTagble
   RUNG wire#powerrail
      { S7_Templates := "SrcType := DInt" } EQ_Contact(in1 := "Unit1.Em5.ControlNodes".gaugeRnR.sequence.status.currentStep, in2 := #JOB_24_STEP_10)
      Contact( "Unit1.Em5.ControlNodes".gaugeRnR.sequence.status.seqActive )
      wire#w1
      Coil( "Unit1.Em5.ControlNodes".gaugeRnR."step".action1[2410] )
   END_RUNG
   RUNG wire#w1
      Contact( "Unit1.Em5.ControlNodes".cm.softCam.cathodeMainPnP1AxisZ.ailgnTableDownPos.inPos )
      Coil( "Unit1.Em5.ControlNodes".gaugeRnR."step".transition1[2410] )
   END_RUNG
   RUNG wire#w1
      Contact( "Unit1.Em5.ControlNodes".gaugeRnR."step".transition1[2410] )
      Move(in := #JOB_24_STEP_20, out1 => "Unit1.Em5.ControlNodes".gaugeRnR.sequence.status.nextStep)
   END_RUNG
   // the same network as SCL:
   "Unit1.Em5.ControlNodes".gaugeRnR."step".action1[2410] := ("Unit1.Em5.ControlNodes".gaugeRnR.sequence.status.currentStep = #JOB_24_STEP_10) AND "Unit1.Em5.ControlNodes".gaugeRnR.sequence.status.seqActive;
   "Unit1.Em5.ControlNodes".gaugeRnR."step".transition1[2410] := ("Unit1.Em5.ControlNodes".gaugeRnR.sequence.status.currentStep = #JOB_24_STEP_10) AND "Unit1.Em5.ControlNodes".gaugeRnR.sequence.status.seqActive AND "Unit1.Em5.ControlNodes".cm.softCam.cathodeMainPnP1AxisZ.ailgnTableDownPos.inPos;
   IF ("Unit1.Em5.ControlNodes".gaugeRnR.sequence.status.currentStep = #JOB_24_STEP_10) AND "Unit1.Em5.ControlNodes".gaugeRnR.sequence.status.seqActive AND "Unit1.Em5.ControlNodes".gaugeRnR."step".transition1[2410] THEN
       "Unit1.Em5.ControlNodes".gaugeRnR.sequence.status.nextStep := #JOB_24_STEP_20;
   END_IF;
END_REGION

REGION Network 120: Step[2420] : AlignTable Vaccum Off
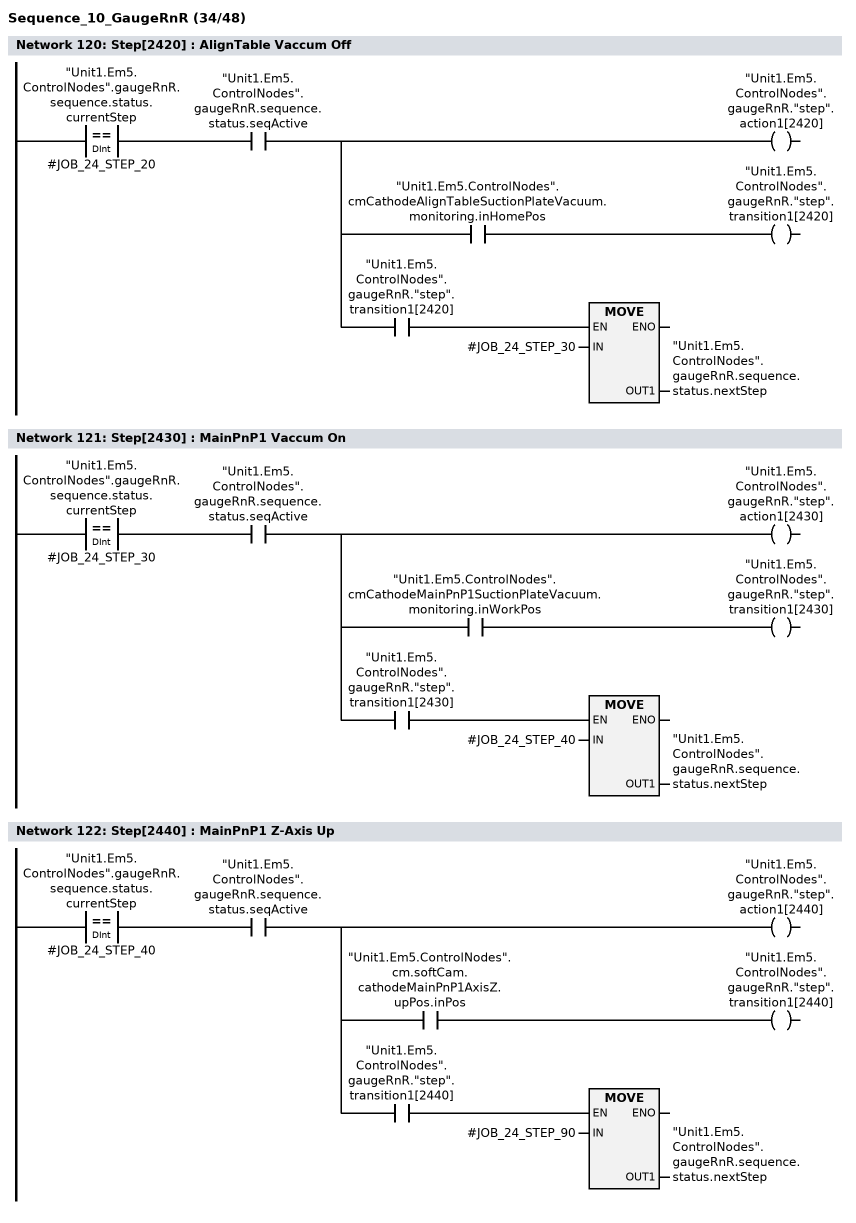
   RUNG wire#powerrail
      { S7_Templates := "SrcType := DInt" } EQ_Contact(in1 := "Unit1.Em5.ControlNodes".gaugeRnR.sequence.status.currentStep, in2 := #JOB_24_STEP_20)
      Contact( "Unit1.Em5.ControlNodes".gaugeRnR.sequence.status.seqActive )
      wire#w1
      Coil( "Unit1.Em5.ControlNodes".gaugeRnR."step".action1[2420] )
   END_RUNG
   RUNG wire#w1
      Contact( "Unit1.Em5.ControlNodes".cmCathodeAlignTableSuctionPlateVacuum.monitoring.inHomePos )
      Coil( "Unit1.Em5.ControlNodes".gaugeRnR."step".transition1[2420] )
   END_RUNG
   RUNG wire#w1
      Contact( "Unit1.Em5.ControlNodes".gaugeRnR."step".transition1[2420] )
      Move(in := #JOB_24_STEP_30, out1 => "Unit1.Em5.ControlNodes".gaugeRnR.sequence.status.nextStep)
   END_RUNG
   // the same network as SCL:
   "Unit1.Em5.ControlNodes".gaugeRnR."step".action1[2420] := ("Unit1.Em5.ControlNodes".gaugeRnR.sequence.status.currentStep = #JOB_24_STEP_20) AND "Unit1.Em5.ControlNodes".gaugeRnR.sequence.status.seqActive;
   "Unit1.Em5.ControlNodes".gaugeRnR."step".transition1[2420] := ("Unit1.Em5.ControlNodes".gaugeRnR.sequence.status.currentStep = #JOB_24_STEP_20) AND "Unit1.Em5.ControlNodes".gaugeRnR.sequence.status.seqActive AND "Unit1.Em5.ControlNodes".cmCathodeAlignTableSuctionPlateVacuum.monitoring.inHomePos;
   IF ("Unit1.Em5.ControlNodes".gaugeRnR.sequence.status.currentStep = #JOB_24_STEP_20) AND "Unit1.Em5.ControlNodes".gaugeRnR.sequence.status.seqActive AND "Unit1.Em5.ControlNodes".gaugeRnR."step".transition1[2420] THEN
       "Unit1.Em5.ControlNodes".gaugeRnR.sequence.status.nextStep := #JOB_24_STEP_30;
   END_IF;
END_REGION

REGION Network 121: Step[2430] : MainPnP1 Vaccum On
   RUNG wire#powerrail
      { S7_Templates := "SrcType := DInt" } EQ_Contact(in1 := "Unit1.Em5.ControlNodes".gaugeRnR.sequence.status.currentStep, in2 := #JOB_24_STEP_30)
      Contact( "Unit1.Em5.ControlNodes".gaugeRnR.sequence.status.seqActive )
      wire#w1
      Coil( "Unit1.Em5.ControlNodes".gaugeRnR."step".action1[2430] )
   END_RUNG
   RUNG wire#w1
      Contact( "Unit1.Em5.ControlNodes".cmCathodeMainPnP1SuctionPlateVacuum.monitoring.inWorkPos )
      Coil( "Unit1.Em5.ControlNodes".gaugeRnR."step".transition1[2430] )
   END_RUNG
   RUNG wire#w1
      Contact( "Unit1.Em5.ControlNodes".gaugeRnR."step".transition1[2430] )
      Move(in := #JOB_24_STEP_40, out1 => "Unit1.Em5.ControlNodes".gaugeRnR.sequence.status.nextStep)
   END_RUNG
   // the same network as SCL:
   "Unit1.Em5.ControlNodes".gaugeRnR."step".action1[2430] := ("Unit1.Em5.ControlNodes".gaugeRnR.sequence.status.currentStep = #JOB_24_STEP_30) AND "Unit1.Em5.ControlNodes".gaugeRnR.sequence.status.seqActive;
   "Unit1.Em5.ControlNodes".gaugeRnR."step".transition1[2430] := ("Unit1.Em5.ControlNodes".gaugeRnR.sequence.status.currentStep = #JOB_24_STEP_30) AND "Unit1.Em5.ControlNodes".gaugeRnR.sequence.status.seqActive AND "Unit1.Em5.ControlNodes".cmCathodeMainPnP1SuctionPlateVacuum.monitoring.inWorkPos;
   IF ("Unit1.Em5.ControlNodes".gaugeRnR.sequence.status.currentStep = #JOB_24_STEP_30) AND "Unit1.Em5.ControlNodes".gaugeRnR.sequence.status.seqActive AND "Unit1.Em5.ControlNodes".gaugeRnR."step".transition1[2430] THEN
       "Unit1.Em5.ControlNodes".gaugeRnR.sequence.status.nextStep := #JOB_24_STEP_40;
   END_IF;
END_REGION

REGION Network 122: Step[2440] : MainPnP1 Z-Axis Up
   RUNG wire#powerrail
      { S7_Templates := "SrcType := DInt" } EQ_Contact(in1 := "Unit1.Em5.ControlNodes".gaugeRnR.sequence.status.currentStep, in2 := #JOB_24_STEP_40)
      Contact( "Unit1.Em5.ControlNodes".gaugeRnR.sequence.status.seqActive )
      wire#w1
      Coil( "Unit1.Em5.ControlNodes".gaugeRnR."step".action1[2440] )
   END_RUNG
   RUNG wire#w1
      Contact( "Unit1.Em5.ControlNodes".cm.softCam.cathodeMainPnP1AxisZ.upPos.inPos )
      Coil( "Unit1.Em5.ControlNodes".gaugeRnR."step".transition1[2440] )
   END_RUNG
   RUNG wire#w1
      Contact( "Unit1.Em5.ControlNodes".gaugeRnR."step".transition1[2440] )
      Move(in := #JOB_24_STEP_90, out1 => "Unit1.Em5.ControlNodes".gaugeRnR.sequence.status.nextStep)
   END_RUNG
   // the same network as SCL:
   "Unit1.Em5.ControlNodes".gaugeRnR."step".action1[2440] := ("Unit1.Em5.ControlNodes".gaugeRnR.sequence.status.currentStep = #JOB_24_STEP_40) AND "Unit1.Em5.ControlNodes".gaugeRnR.sequence.status.seqActive;
   "Unit1.Em5.ControlNodes".gaugeRnR."step".transition1[2440] := ("Unit1.Em5.ControlNodes".gaugeRnR.sequence.status.currentStep = #JOB_24_STEP_40) AND "Unit1.Em5.ControlNodes".gaugeRnR.sequence.status.seqActive AND "Unit1.Em5.ControlNodes".cm.softCam.cathodeMainPnP1AxisZ.upPos.inPos;
   IF ("Unit1.Em5.ControlNodes".gaugeRnR.sequence.status.currentStep = #JOB_24_STEP_40) AND "Unit1.Em5.ControlNodes".gaugeRnR.sequence.status.seqActive AND "Unit1.Em5.ControlNodes".gaugeRnR."step".transition1[2440] THEN
       "Unit1.Em5.ControlNodes".gaugeRnR.sequence.status.nextStep := #JOB_24_STEP_90;
   END_IF;
END_REGION

REGION Network 123: Step[2490] : Job[10] Step End
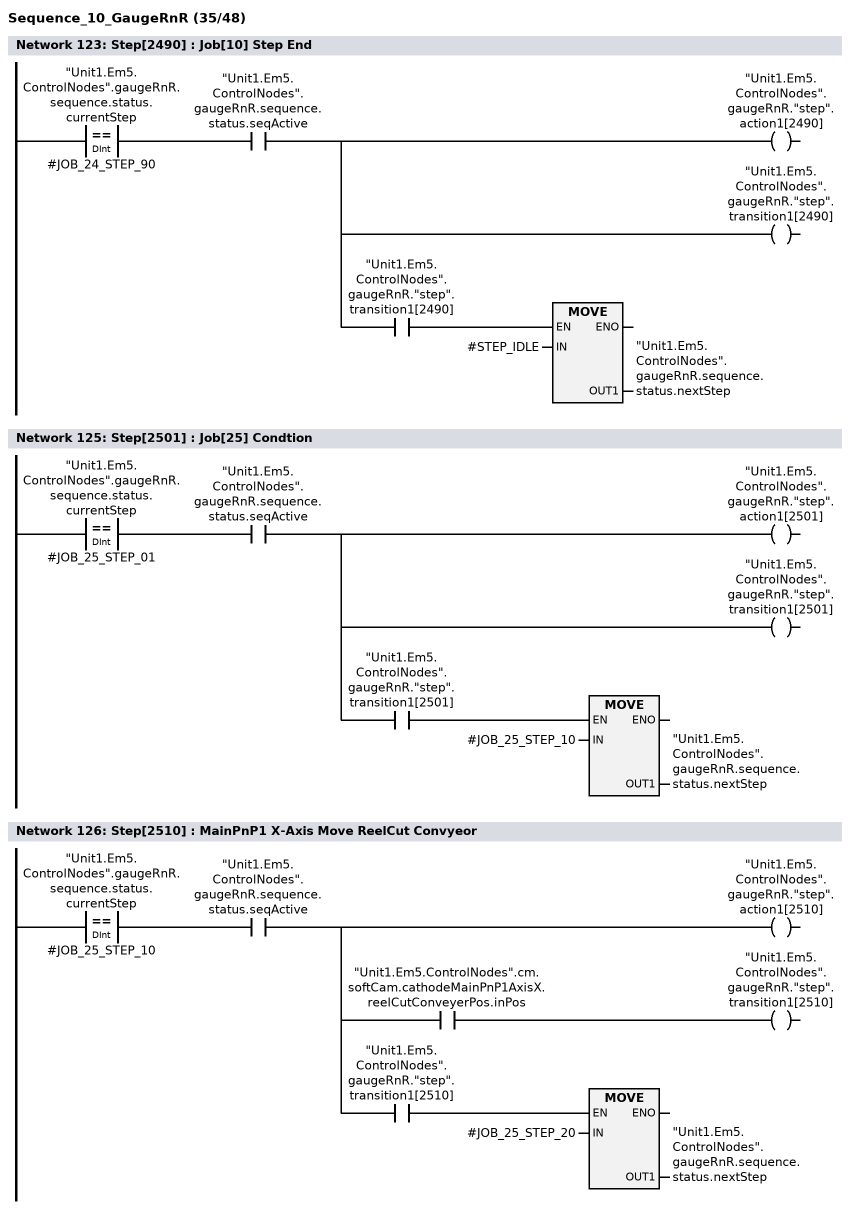
   RUNG wire#powerrail
      { S7_Templates := "SrcType := DInt" } EQ_Contact(in1 := "Unit1.Em5.ControlNodes".gaugeRnR.sequence.status.currentStep, in2 := #JOB_24_STEP_90)
      Contact( "Unit1.Em5.ControlNodes".gaugeRnR.sequence.status.seqActive )
      wire#w1
      Coil( "Unit1.Em5.ControlNodes".gaugeRnR."step".action1[2490] )
   END_RUNG
   RUNG wire#w1
      Coil( "Unit1.Em5.ControlNodes".gaugeRnR."step".transition1[2490] )
   END_RUNG
   RUNG wire#w1
      Contact( "Unit1.Em5.ControlNodes".gaugeRnR."step".transition1[2490] )
      Move(in := #STEP_IDLE, out1 => "Unit1.Em5.ControlNodes".gaugeRnR.sequence.status.nextStep)
   END_RUNG
   // the same network as SCL:
   "Unit1.Em5.ControlNodes".gaugeRnR."step".action1[2490] := ("Unit1.Em5.ControlNodes".gaugeRnR.sequence.status.currentStep = #JOB_24_STEP_90) AND "Unit1.Em5.ControlNodes".gaugeRnR.sequence.status.seqActive;
   "Unit1.Em5.ControlNodes".gaugeRnR."step".transition1[2490] := ("Unit1.Em5.ControlNodes".gaugeRnR.sequence.status.currentStep = #JOB_24_STEP_90) AND "Unit1.Em5.ControlNodes".gaugeRnR.sequence.status.seqActive;
   IF ("Unit1.Em5.ControlNodes".gaugeRnR.sequence.status.currentStep = #JOB_24_STEP_90) AND "Unit1.Em5.ControlNodes".gaugeRnR.sequence.status.seqActive AND "Unit1.Em5.ControlNodes".gaugeRnR."step".transition1[2490] THEN
       "Unit1.Em5.ControlNodes".gaugeRnR.sequence.status.nextStep := #STEP_IDLE;
   END_IF;
END_REGION

REGION Network 124: *************** JOB[25] MainPnP Move ReelCut Convyeor / AlignTable************************
END_REGION

REGION Network 125: Step[2501] : Job[25] Condtion
   RUNG wire#powerrail
      { S7_Templates := "SrcType := DInt" } EQ_Contact(in1 := "Unit1.Em5.ControlNodes".gaugeRnR.sequence.status.currentStep, in2 := #JOB_25_STEP_01)
      Contact( "Unit1.Em5.ControlNodes".gaugeRnR.sequence.status.seqActive )
      wire#w1
      Coil( "Unit1.Em5.ControlNodes".gaugeRnR."step".action1[2501] )
   END_RUNG
   RUNG wire#w1
      Coil( "Unit1.Em5.ControlNodes".gaugeRnR."step".transition1[2501] )
   END_RUNG
   RUNG wire#w1
      Contact( "Unit1.Em5.ControlNodes".gaugeRnR."step".transition1[2501] )
      Move(in := #JOB_25_STEP_10, out1 => "Unit1.Em5.ControlNodes".gaugeRnR.sequence.status.nextStep)
   END_RUNG
   // the same network as SCL:
   "Unit1.Em5.ControlNodes".gaugeRnR."step".action1[2501] := ("Unit1.Em5.ControlNodes".gaugeRnR.sequence.status.currentStep = #JOB_25_STEP_01) AND "Unit1.Em5.ControlNodes".gaugeRnR.sequence.status.seqActive;
   "Unit1.Em5.ControlNodes".gaugeRnR."step".transition1[2501] := ("Unit1.Em5.ControlNodes".gaugeRnR.sequence.status.currentStep = #JOB_25_STEP_01) AND "Unit1.Em5.ControlNodes".gaugeRnR.sequence.status.seqActive;
   IF ("Unit1.Em5.ControlNodes".gaugeRnR.sequence.status.currentStep = #JOB_25_STEP_01) AND "Unit1.Em5.ControlNodes".gaugeRnR.sequence.status.seqActive AND "Unit1.Em5.ControlNodes".gaugeRnR."step".transition1[2501] THEN
       "Unit1.Em5.ControlNodes".gaugeRnR.sequence.status.nextStep := #JOB_25_STEP_10;
   END_IF;
END_REGION

REGION Network 126: Step[2510] : MainPnP1 X-Axis Move ReelCut Convyeor
   RUNG wire#powerrail
      { S7_Templates := "SrcType := DInt" } EQ_Contact(in1 := "Unit1.Em5.ControlNodes".gaugeRnR.sequence.status.currentStep, in2 := #JOB_25_STEP_10)
      Contact( "Unit1.Em5.ControlNodes".gaugeRnR.sequence.status.seqActive )
      wire#w1
      Coil( "Unit1.Em5.ControlNodes".gaugeRnR."step".action1[2510] )
   END_RUNG
   RUNG wire#w1
      Contact( "Unit1.Em5.ControlNodes".cm.softCam.cathodeMainPnP1AxisX.reelCutConveyerPos.inPos )
      Coil( "Unit1.Em5.ControlNodes".gaugeRnR."step".transition1[2510] )
   END_RUNG
   RUNG wire#w1
      Contact( "Unit1.Em5.ControlNodes".gaugeRnR."step".transition1[2510] )
      Move(in := #JOB_25_STEP_20, out1 => "Unit1.Em5.ControlNodes".gaugeRnR.sequence.status.nextStep)
   END_RUNG
   // the same network as SCL:
   "Unit1.Em5.ControlNodes".gaugeRnR."step".action1[2510] := ("Unit1.Em5.ControlNodes".gaugeRnR.sequence.status.currentStep = #JOB_25_STEP_10) AND "Unit1.Em5.ControlNodes".gaugeRnR.sequence.status.seqActive;
   "Unit1.Em5.ControlNodes".gaugeRnR."step".transition1[2510] := ("Unit1.Em5.ControlNodes".gaugeRnR.sequence.status.currentStep = #JOB_25_STEP_10) AND "Unit1.Em5.ControlNodes".gaugeRnR.sequence.status.seqActive AND "Unit1.Em5.ControlNodes".cm.softCam.cathodeMainPnP1AxisX.reelCutConveyerPos.inPos;
   IF ("Unit1.Em5.ControlNodes".gaugeRnR.sequence.status.currentStep = #JOB_25_STEP_10) AND "Unit1.Em5.ControlNodes".gaugeRnR.sequence.status.seqActive AND "Unit1.Em5.ControlNodes".gaugeRnR."step".transition1[2510] THEN
       "Unit1.Em5.ControlNodes".gaugeRnR.sequence.status.nextStep := #JOB_25_STEP_20;
   END_IF;
END_REGION

REGION Network 127: Step[2520] : MainPnP2 X-Axis Move AlignTable
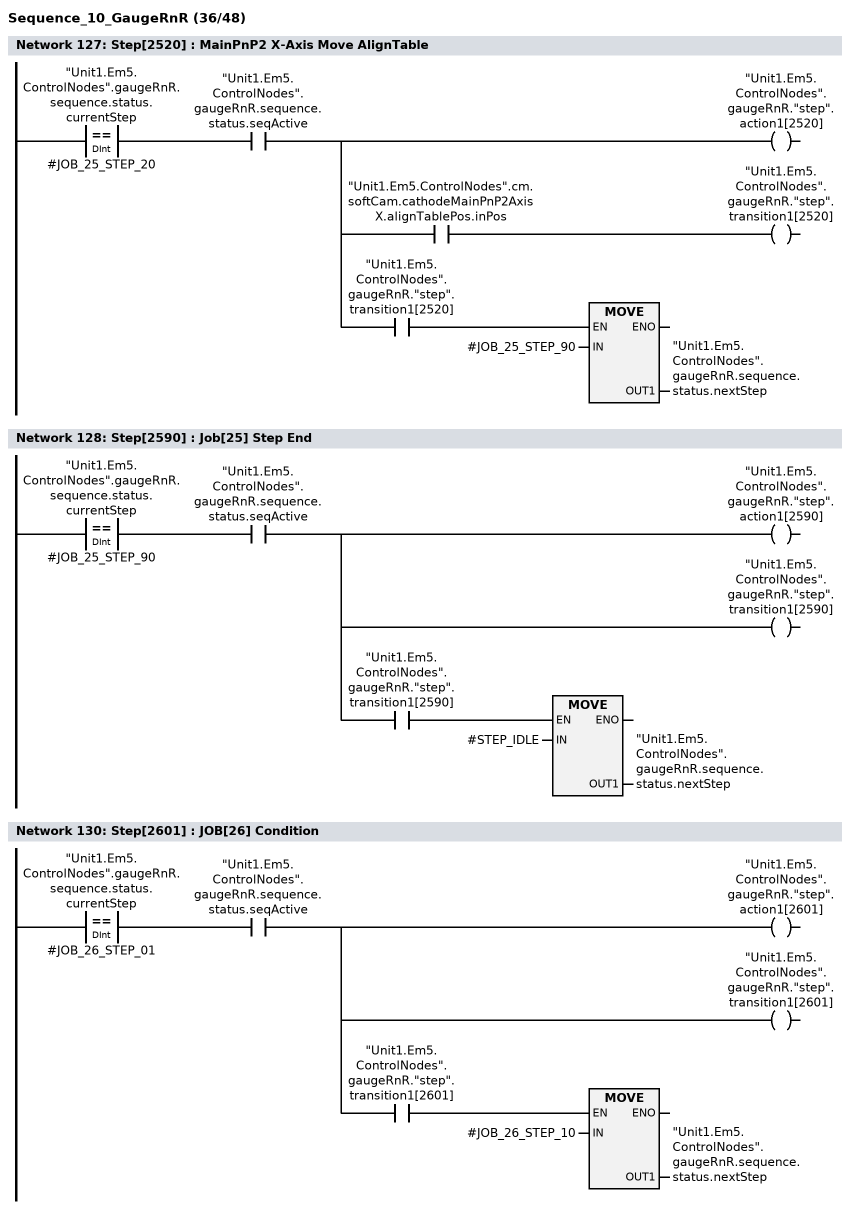
   RUNG wire#powerrail
      { S7_Templates := "SrcType := DInt" } EQ_Contact(in1 := "Unit1.Em5.ControlNodes".gaugeRnR.sequence.status.currentStep, in2 := #JOB_25_STEP_20)
      Contact( "Unit1.Em5.ControlNodes".gaugeRnR.sequence.status.seqActive )
      wire#w1
      Coil( "Unit1.Em5.ControlNodes".gaugeRnR."step".action1[2520] )
   END_RUNG
   RUNG wire#w1
      Contact( "Unit1.Em5.ControlNodes".cm.softCam.cathodeMainPnP2AxisX.alignTablePos.inPos )
      Coil( "Unit1.Em5.ControlNodes".gaugeRnR."step".transition1[2520] )
   END_RUNG
   RUNG wire#w1
      Contact( "Unit1.Em5.ControlNodes".gaugeRnR."step".transition1[2520] )
      Move(in := #JOB_25_STEP_90, out1 => "Unit1.Em5.ControlNodes".gaugeRnR.sequence.status.nextStep)
   END_RUNG
   // the same network as SCL:
   "Unit1.Em5.ControlNodes".gaugeRnR."step".action1[2520] := ("Unit1.Em5.ControlNodes".gaugeRnR.sequence.status.currentStep = #JOB_25_STEP_20) AND "Unit1.Em5.ControlNodes".gaugeRnR.sequence.status.seqActive;
   "Unit1.Em5.ControlNodes".gaugeRnR."step".transition1[2520] := ("Unit1.Em5.ControlNodes".gaugeRnR.sequence.status.currentStep = #JOB_25_STEP_20) AND "Unit1.Em5.ControlNodes".gaugeRnR.sequence.status.seqActive AND "Unit1.Em5.ControlNodes".cm.softCam.cathodeMainPnP2AxisX.alignTablePos.inPos;
   IF ("Unit1.Em5.ControlNodes".gaugeRnR.sequence.status.currentStep = #JOB_25_STEP_20) AND "Unit1.Em5.ControlNodes".gaugeRnR.sequence.status.seqActive AND "Unit1.Em5.ControlNodes".gaugeRnR."step".transition1[2520] THEN
       "Unit1.Em5.ControlNodes".gaugeRnR.sequence.status.nextStep := #JOB_25_STEP_90;
   END_IF;
END_REGION

REGION Network 128: Step[2590] : Job[25] Step End
   RUNG wire#powerrail
      { S7_Templates := "SrcType := DInt" } EQ_Contact(in1 := "Unit1.Em5.ControlNodes".gaugeRnR.sequence.status.currentStep, in2 := #JOB_25_STEP_90)
      Contact( "Unit1.Em5.ControlNodes".gaugeRnR.sequence.status.seqActive )
      wire#w1
      Coil( "Unit1.Em5.ControlNodes".gaugeRnR."step".action1[2590] )
   END_RUNG
   RUNG wire#w1
      Coil( "Unit1.Em5.ControlNodes".gaugeRnR."step".transition1[2590] )
   END_RUNG
   RUNG wire#w1
      Contact( "Unit1.Em5.ControlNodes".gaugeRnR."step".transition1[2590] )
      Move(in := #STEP_IDLE, out1 => "Unit1.Em5.ControlNodes".gaugeRnR.sequence.status.nextStep)
   END_RUNG
   // the same network as SCL:
   "Unit1.Em5.ControlNodes".gaugeRnR."step".action1[2590] := ("Unit1.Em5.ControlNodes".gaugeRnR.sequence.status.currentStep = #JOB_25_STEP_90) AND "Unit1.Em5.ControlNodes".gaugeRnR.sequence.status.seqActive;
   "Unit1.Em5.ControlNodes".gaugeRnR."step".transition1[2590] := ("Unit1.Em5.ControlNodes".gaugeRnR.sequence.status.currentStep = #JOB_25_STEP_90) AND "Unit1.Em5.ControlNodes".gaugeRnR.sequence.status.seqActive;
   IF ("Unit1.Em5.ControlNodes".gaugeRnR.sequence.status.currentStep = #JOB_25_STEP_90) AND "Unit1.Em5.ControlNodes".gaugeRnR.sequence.status.seqActive AND "Unit1.Em5.ControlNodes".gaugeRnR."step".transition1[2590] THEN
       "Unit1.Em5.ControlNodes".gaugeRnR.sequence.status.nextStep := #STEP_IDLE;
   END_IF;
END_REGION

REGION Network 129: *************** JOB[26] Unload MasterPiece ************************
END_REGION

REGION Network 130: Step[2601] : JOB[26] Condition
   RUNG wire#powerrail
      { S7_Templates := "SrcType := DInt" } EQ_Contact(in1 := "Unit1.Em5.ControlNodes".gaugeRnR.sequence.status.currentStep, in2 := #JOB_26_STEP_01)
      Contact( "Unit1.Em5.ControlNodes".gaugeRnR.sequence.status.seqActive )
      wire#w1
      Coil( "Unit1.Em5.ControlNodes".gaugeRnR."step".action1[2601] )
   END_RUNG
   RUNG wire#w1
      Coil( "Unit1.Em5.ControlNodes".gaugeRnR."step".transition1[2601] )
   END_RUNG
   RUNG wire#w1
      Contact( "Unit1.Em5.ControlNodes".gaugeRnR."step".transition1[2601] )
      Move(in := #JOB_26_STEP_10, out1 => "Unit1.Em5.ControlNodes".gaugeRnR.sequence.status.nextStep)
   END_RUNG
   // the same network as SCL:
   "Unit1.Em5.ControlNodes".gaugeRnR."step".action1[2601] := ("Unit1.Em5.ControlNodes".gaugeRnR.sequence.status.currentStep = #JOB_26_STEP_01) AND "Unit1.Em5.ControlNodes".gaugeRnR.sequence.status.seqActive;
   "Unit1.Em5.ControlNodes".gaugeRnR."step".transition1[2601] := ("Unit1.Em5.ControlNodes".gaugeRnR.sequence.status.currentStep = #JOB_26_STEP_01) AND "Unit1.Em5.ControlNodes".gaugeRnR.sequence.status.seqActive;
   IF ("Unit1.Em5.ControlNodes".gaugeRnR.sequence.status.currentStep = #JOB_26_STEP_01) AND "Unit1.Em5.ControlNodes".gaugeRnR.sequence.status.seqActive AND "Unit1.Em5.ControlNodes".gaugeRnR."step".transition1[2601] THEN
       "Unit1.Em5.ControlNodes".gaugeRnR.sequence.status.nextStep := #JOB_26_STEP_10;
   END_IF;
END_REGION

REGION Network 131: Step[2610] : MainPnP1 Z-Axis Conveyor Down
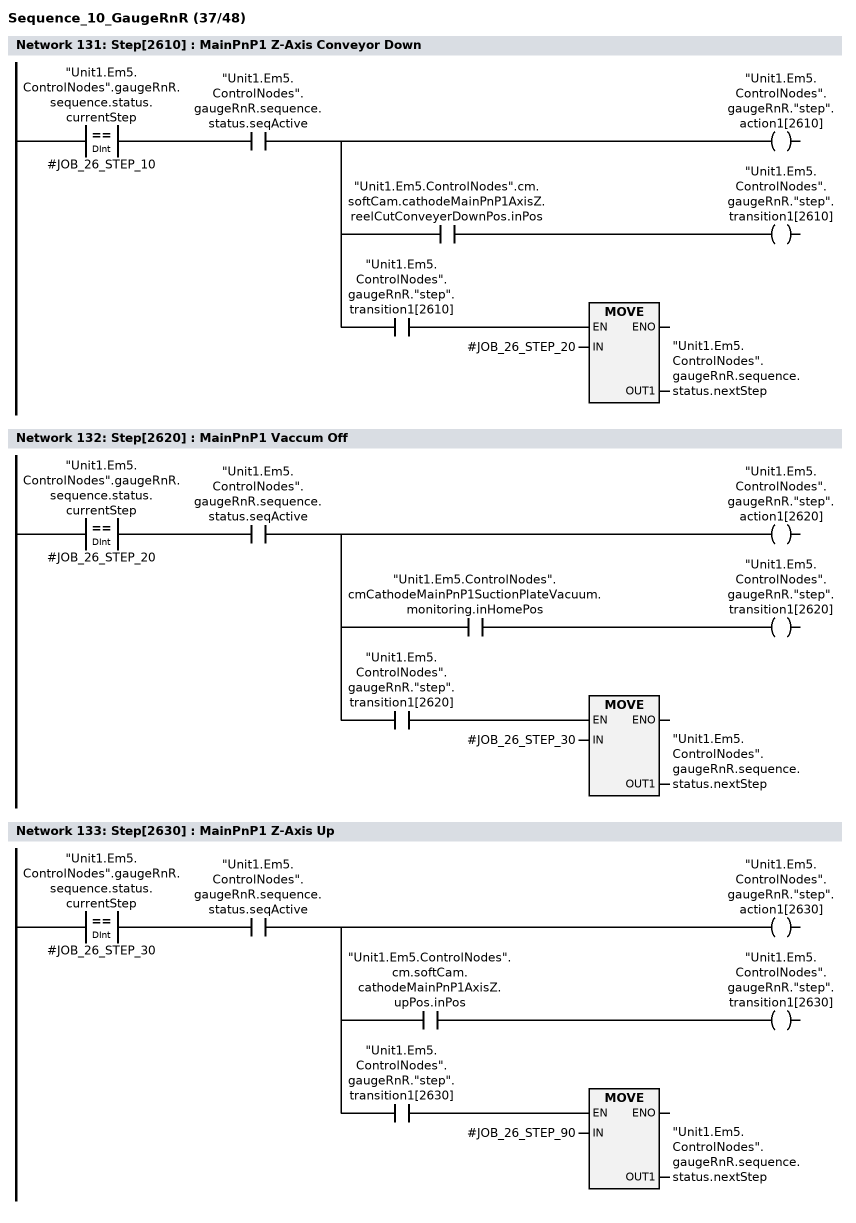
   RUNG wire#powerrail
      { S7_Templates := "SrcType := DInt" } EQ_Contact(in1 := "Unit1.Em5.ControlNodes".gaugeRnR.sequence.status.currentStep, in2 := #JOB_26_STEP_10)
      Contact( "Unit1.Em5.ControlNodes".gaugeRnR.sequence.status.seqActive )
      wire#w1
      Coil( "Unit1.Em5.ControlNodes".gaugeRnR."step".action1[2610] )
   END_RUNG
   RUNG wire#w1
      Contact( "Unit1.Em5.ControlNodes".cm.softCam.cathodeMainPnP1AxisZ.reelCutConveyerDownPos.inPos )
      Coil( "Unit1.Em5.ControlNodes".gaugeRnR."step".transition1[2610] )
   END_RUNG
   RUNG wire#w1
      Contact( "Unit1.Em5.ControlNodes".gaugeRnR."step".transition1[2610] )
      Move(in := #JOB_26_STEP_20, out1 => "Unit1.Em5.ControlNodes".gaugeRnR.sequence.status.nextStep)
   END_RUNG
   // the same network as SCL:
   "Unit1.Em5.ControlNodes".gaugeRnR."step".action1[2610] := ("Unit1.Em5.ControlNodes".gaugeRnR.sequence.status.currentStep = #JOB_26_STEP_10) AND "Unit1.Em5.ControlNodes".gaugeRnR.sequence.status.seqActive;
   "Unit1.Em5.ControlNodes".gaugeRnR."step".transition1[2610] := ("Unit1.Em5.ControlNodes".gaugeRnR.sequence.status.currentStep = #JOB_26_STEP_10) AND "Unit1.Em5.ControlNodes".gaugeRnR.sequence.status.seqActive AND "Unit1.Em5.ControlNodes".cm.softCam.cathodeMainPnP1AxisZ.reelCutConveyerDownPos.inPos;
   IF ("Unit1.Em5.ControlNodes".gaugeRnR.sequence.status.currentStep = #JOB_26_STEP_10) AND "Unit1.Em5.ControlNodes".gaugeRnR.sequence.status.seqActive AND "Unit1.Em5.ControlNodes".gaugeRnR."step".transition1[2610] THEN
       "Unit1.Em5.ControlNodes".gaugeRnR.sequence.status.nextStep := #JOB_26_STEP_20;
   END_IF;
END_REGION

REGION Network 132: Step[2620] : MainPnP1 Vaccum Off
   RUNG wire#powerrail
      { S7_Templates := "SrcType := DInt" } EQ_Contact(in1 := "Unit1.Em5.ControlNodes".gaugeRnR.sequence.status.currentStep, in2 := #JOB_26_STEP_20)
      Contact( "Unit1.Em5.ControlNodes".gaugeRnR.sequence.status.seqActive )
      wire#w1
      Coil( "Unit1.Em5.ControlNodes".gaugeRnR."step".action1[2620] )
   END_RUNG
   RUNG wire#w1
      Contact( "Unit1.Em5.ControlNodes".cmCathodeMainPnP1SuctionPlateVacuum.monitoring.inHomePos )
      Coil( "Unit1.Em5.ControlNodes".gaugeRnR."step".transition1[2620] )
   END_RUNG
   RUNG wire#w1
      Contact( "Unit1.Em5.ControlNodes".gaugeRnR."step".transition1[2620] )
      Move(in := #JOB_26_STEP_30, out1 => "Unit1.Em5.ControlNodes".gaugeRnR.sequence.status.nextStep)
   END_RUNG
   // the same network as SCL:
   "Unit1.Em5.ControlNodes".gaugeRnR."step".action1[2620] := ("Unit1.Em5.ControlNodes".gaugeRnR.sequence.status.currentStep = #JOB_26_STEP_20) AND "Unit1.Em5.ControlNodes".gaugeRnR.sequence.status.seqActive;
   "Unit1.Em5.ControlNodes".gaugeRnR."step".transition1[2620] := ("Unit1.Em5.ControlNodes".gaugeRnR.sequence.status.currentStep = #JOB_26_STEP_20) AND "Unit1.Em5.ControlNodes".gaugeRnR.sequence.status.seqActive AND "Unit1.Em5.ControlNodes".cmCathodeMainPnP1SuctionPlateVacuum.monitoring.inHomePos;
   IF ("Unit1.Em5.ControlNodes".gaugeRnR.sequence.status.currentStep = #JOB_26_STEP_20) AND "Unit1.Em5.ControlNodes".gaugeRnR.sequence.status.seqActive AND "Unit1.Em5.ControlNodes".gaugeRnR."step".transition1[2620] THEN
       "Unit1.Em5.ControlNodes".gaugeRnR.sequence.status.nextStep := #JOB_26_STEP_30;
   END_IF;
END_REGION

REGION Network 133: Step[2630] : MainPnP1 Z-Axis Up
   RUNG wire#powerrail
      { S7_Templates := "SrcType := DInt" } EQ_Contact(in1 := "Unit1.Em5.ControlNodes".gaugeRnR.sequence.status.currentStep, in2 := #JOB_26_STEP_30)
      Contact( "Unit1.Em5.ControlNodes".gaugeRnR.sequence.status.seqActive )
      wire#w1
      Coil( "Unit1.Em5.ControlNodes".gaugeRnR."step".action1[2630] )
   END_RUNG
   RUNG wire#w1
      Contact( "Unit1.Em5.ControlNodes".cm.softCam.cathodeMainPnP1AxisZ.upPos.inPos )
      Coil( "Unit1.Em5.ControlNodes".gaugeRnR."step".transition1[2630] )
   END_RUNG
   RUNG wire#w1
      Contact( "Unit1.Em5.ControlNodes".gaugeRnR."step".transition1[2630] )
      Move(in := #JOB_26_STEP_90, out1 => "Unit1.Em5.ControlNodes".gaugeRnR.sequence.status.nextStep)
   END_RUNG
   // the same network as SCL:
   "Unit1.Em5.ControlNodes".gaugeRnR."step".action1[2630] := ("Unit1.Em5.ControlNodes".gaugeRnR.sequence.status.currentStep = #JOB_26_STEP_30) AND "Unit1.Em5.ControlNodes".gaugeRnR.sequence.status.seqActive;
   "Unit1.Em5.ControlNodes".gaugeRnR."step".transition1[2630] := ("Unit1.Em5.ControlNodes".gaugeRnR.sequence.status.currentStep = #JOB_26_STEP_30) AND "Unit1.Em5.ControlNodes".gaugeRnR.sequence.status.seqActive AND "Unit1.Em5.ControlNodes".cm.softCam.cathodeMainPnP1AxisZ.upPos.inPos;
   IF ("Unit1.Em5.ControlNodes".gaugeRnR.sequence.status.currentStep = #JOB_26_STEP_30) AND "Unit1.Em5.ControlNodes".gaugeRnR.sequence.status.seqActive AND "Unit1.Em5.ControlNodes".gaugeRnR."step".transition1[2630] THEN
       "Unit1.Em5.ControlNodes".gaugeRnR.sequence.status.nextStep := #JOB_26_STEP_90;
   END_IF;
END_REGION

REGION Network 134: Step[2690] : Job[26] Step End
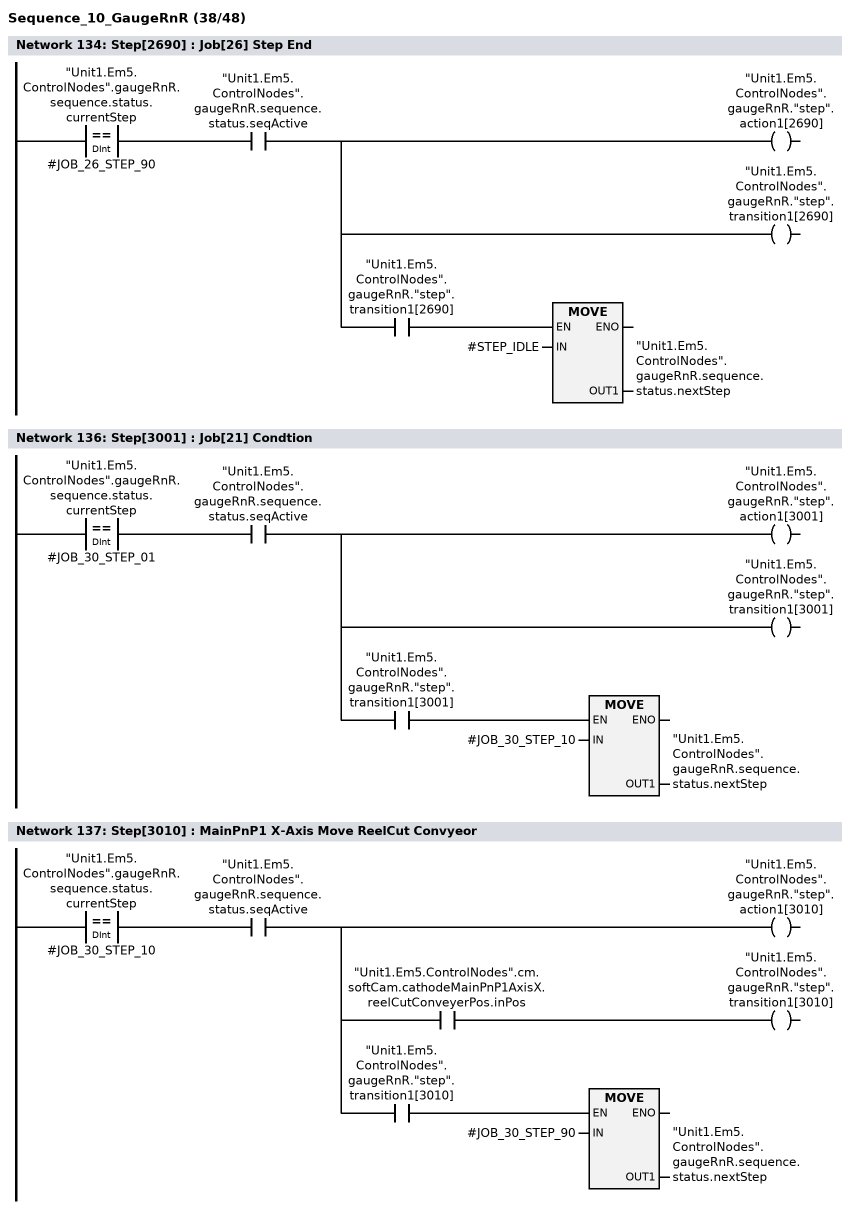
   RUNG wire#powerrail
      { S7_Templates := "SrcType := DInt" } EQ_Contact(in1 := "Unit1.Em5.ControlNodes".gaugeRnR.sequence.status.currentStep, in2 := #JOB_26_STEP_90)
      Contact( "Unit1.Em5.ControlNodes".gaugeRnR.sequence.status.seqActive )
      wire#w1
      Coil( "Unit1.Em5.ControlNodes".gaugeRnR."step".action1[2690] )
   END_RUNG
   RUNG wire#w1
      Coil( "Unit1.Em5.ControlNodes".gaugeRnR."step".transition1[2690] )
   END_RUNG
   RUNG wire#w1
      Contact( "Unit1.Em5.ControlNodes".gaugeRnR."step".transition1[2690] )
      Move(in := #STEP_IDLE, out1 => "Unit1.Em5.ControlNodes".gaugeRnR.sequence.status.nextStep)
   END_RUNG
   // the same network as SCL:
   "Unit1.Em5.ControlNodes".gaugeRnR."step".action1[2690] := ("Unit1.Em5.ControlNodes".gaugeRnR.sequence.status.currentStep = #JOB_26_STEP_90) AND "Unit1.Em5.ControlNodes".gaugeRnR.sequence.status.seqActive;
   "Unit1.Em5.ControlNodes".gaugeRnR."step".transition1[2690] := ("Unit1.Em5.ControlNodes".gaugeRnR.sequence.status.currentStep = #JOB_26_STEP_90) AND "Unit1.Em5.ControlNodes".gaugeRnR.sequence.status.seqActive;
   IF ("Unit1.Em5.ControlNodes".gaugeRnR.sequence.status.currentStep = #JOB_26_STEP_90) AND "Unit1.Em5.ControlNodes".gaugeRnR.sequence.status.seqActive AND "Unit1.Em5.ControlNodes".gaugeRnR."step".transition1[2690] THEN
       "Unit1.Em5.ControlNodes".gaugeRnR.sequence.status.nextStep := #STEP_IDLE;
   END_IF;
END_REGION

REGION Network 135: *************** JOB[30] MainPnP1 Move ReelCut Convyeor ************************
END_REGION

REGION Network 136: Step[3001] : Job[21] Condtion
   RUNG wire#powerrail
      { S7_Templates := "SrcType := DInt" } EQ_Contact(in1 := "Unit1.Em5.ControlNodes".gaugeRnR.sequence.status.currentStep, in2 := #JOB_30_STEP_01)
      Contact( "Unit1.Em5.ControlNodes".gaugeRnR.sequence.status.seqActive )
      wire#w1
      Coil( "Unit1.Em5.ControlNodes".gaugeRnR."step".action1[3001] )
   END_RUNG
   RUNG wire#w1
      Coil( "Unit1.Em5.ControlNodes".gaugeRnR."step".transition1[3001] )
   END_RUNG
   RUNG wire#w1
      Contact( "Unit1.Em5.ControlNodes".gaugeRnR."step".transition1[3001] )
      Move(in := #JOB_30_STEP_10, out1 => "Unit1.Em5.ControlNodes".gaugeRnR.sequence.status.nextStep)
   END_RUNG
   // the same network as SCL:
   "Unit1.Em5.ControlNodes".gaugeRnR."step".action1[3001] := ("Unit1.Em5.ControlNodes".gaugeRnR.sequence.status.currentStep = #JOB_30_STEP_01) AND "Unit1.Em5.ControlNodes".gaugeRnR.sequence.status.seqActive;
   "Unit1.Em5.ControlNodes".gaugeRnR."step".transition1[3001] := ("Unit1.Em5.ControlNodes".gaugeRnR.sequence.status.currentStep = #JOB_30_STEP_01) AND "Unit1.Em5.ControlNodes".gaugeRnR.sequence.status.seqActive;
   IF ("Unit1.Em5.ControlNodes".gaugeRnR.sequence.status.currentStep = #JOB_30_STEP_01) AND "Unit1.Em5.ControlNodes".gaugeRnR.sequence.status.seqActive AND "Unit1.Em5.ControlNodes".gaugeRnR."step".transition1[3001] THEN
       "Unit1.Em5.ControlNodes".gaugeRnR.sequence.status.nextStep := #JOB_30_STEP_10;
   END_IF;
END_REGION

REGION Network 137: Step[3010] : MainPnP1 X-Axis Move ReelCut Convyeor
   RUNG wire#powerrail
      { S7_Templates := "SrcType := DInt" } EQ_Contact(in1 := "Unit1.Em5.ControlNodes".gaugeRnR.sequence.status.currentStep, in2 := #JOB_30_STEP_10)
      Contact( "Unit1.Em5.ControlNodes".gaugeRnR.sequence.status.seqActive )
      wire#w1
      Coil( "Unit1.Em5.ControlNodes".gaugeRnR."step".action1[3010] )
   END_RUNG
   RUNG wire#w1
      Contact( "Unit1.Em5.ControlNodes".cm.softCam.cathodeMainPnP1AxisX.reelCutConveyerPos.inPos )
      Coil( "Unit1.Em5.ControlNodes".gaugeRnR."step".transition1[3010] )
   END_RUNG
   RUNG wire#w1
      Contact( "Unit1.Em5.ControlNodes".gaugeRnR."step".transition1[3010] )
      Move(in := #JOB_30_STEP_90, out1 => "Unit1.Em5.ControlNodes".gaugeRnR.sequence.status.nextStep)
   END_RUNG
   // the same network as SCL:
   "Unit1.Em5.ControlNodes".gaugeRnR."step".action1[3010] := ("Unit1.Em5.ControlNodes".gaugeRnR.sequence.status.currentStep = #JOB_30_STEP_10) AND "Unit1.Em5.ControlNodes".gaugeRnR.sequence.status.seqActive;
   "Unit1.Em5.ControlNodes".gaugeRnR."step".transition1[3010] := ("Unit1.Em5.ControlNodes".gaugeRnR.sequence.status.currentStep = #JOB_30_STEP_10) AND "Unit1.Em5.ControlNodes".gaugeRnR.sequence.status.seqActive AND "Unit1.Em5.ControlNodes".cm.softCam.cathodeMainPnP1AxisX.reelCutConveyerPos.inPos;
   IF ("Unit1.Em5.ControlNodes".gaugeRnR.sequence.status.currentStep = #JOB_30_STEP_10) AND "Unit1.Em5.ControlNodes".gaugeRnR.sequence.status.seqActive AND "Unit1.Em5.ControlNodes".gaugeRnR."step".transition1[3010] THEN
       "Unit1.Em5.ControlNodes".gaugeRnR.sequence.status.nextStep := #JOB_30_STEP_90;
   END_IF;
END_REGION

